// TwinCAT 3 PLC project TE1108
// ProgramVersion: 3.1.4026.22
// libraries:
//   Tc2_EtherCAT, * (Beckhoff Automation GmbH)
//   Tc2_IoFunctions, * (Beckhoff Automation GmbH)
//   Tc2_Standard, * (Beckhoff Automation GmbH)
//   Tc2_System, * (Beckhoff Automation GmbH)
//   Tc2_Utilities, * (Beckhoff Automation GmbH)
//   Tc3_Module, * (Beckhoff Automation GmbH)
// project tree:
//   DUTs/COMPONENTS/CAMERA/ ST_Camera.TcDUT, E_Camera_State.TcDUT, ST_Camera_CycleData.TcDUT (not stored), ST_Camera_CMD.TcDUT (not stored)
//   DUTs/COMPONENTS/GENERIC/ ST_GeneralStationCMD.TcDUT (not stored), ST_StationStatus.TcDUT
//   DUTs/COMPONENTS/HEIGHT TEST/ ST_HeightTest.TcDUT, ST_HeightTest_CMD.TcDUT, ST_ProbesSettings.TcDUT, E_HeightTest_State.TcDUT, ST_HeightTest_CycleData.TcDUT (not stored)
//   DUTs/COMPONENTS/LEAK TESTER/ ST_LeakTester.TcDUT, ST_LeakTester_CMD.TcDUT, E_LeakTester_State.TcDUT (not stored), ST_LeakTester_CycleData.TcDUT (not stored)
//   DUTs/COMPONENTS/MAIN CYLINDER/ ST_ProcessCylinder.TcDUT, E_ProcessCylinder_State.TcDUT, ST_ProcessCylinder_CMD.TcDUT (not stored)
//   DUTs/COMPONENTS/PROCESS DOOR/ E_ProcessDoor_State.TcDUT, ST_ProcessDoor.TcDUT, ST_ProcessDoor_CMD.TcDUT
//   DUTs/COMPONENTS/PUCK_LOCKER/ E_PuckLockerMode.TcDUT, E_PuckLockerState.TcDUT, ST_PuckLocker.TcDUT, ST_PuckLockerHMI.TcDUT
//   DUTs/HMI/ ST_Animations.TcDUT, ST_StatisticsHMI.TcDUT, ST_StatusBanner.TcDUT, ST_Timers.TcDUT (not stored)
//   DUTs/IO/CAMERA/ ST_KeyenceCamera_I_O.TcDUT
//   DUTs/IO/CARDS/ ST_EL1918_C.TcDUT, ST_EL3058.TcDUT (not stored), ST_EL1918_A.TcDUT, ST_EL1918_B.TcDUT, ST_EL2904.TcDUT, ST_EL6910.TcDUT, ST_EL6633.TcDUT, ST_EL9410.TcDUT, ST_K1100.TcDUT (not stored), ST_EL6070.TcDUT (not stored), ST_Terminal_Info.TcDUT (not stored), ST_EL1809.TcDUT, ST_EL2809_A.TcDUT
//   DUTs/IO/LEAK_TESTERS/ ST_General_LeakTester_I_O.TcDUT (not stored), st_i28General_I_O.TcDUT, st_i28LasResult.TcDUT, st_i28LiveMeasurement.TcDUT
//   DUTs/IO/PROBES/ ST_ProbesSet.TcDUT, ST_Probes_I_O.TcDUT
//   DUTs/MASTER/ E_MachineState.TcDUT, ST_ButtonsLamps.TcDUT, ST_HMI_IO.TcDUT (not stored), ST_MACHINE.TcDUT, ST_MachineStatus.TcDUT, ST_MasterCTRL.TcDUT, ST_Puls.TcDUT
//   DUTs/MASTER/log_CSV/ ST_TableCycleData.TcDUT (not stored), ST_UserLog.TcDUT, ST_CycleData.TcDUT (not stored)
//   DUTs/MASTER/PROCESS CYCLES/ E_General_ProcessCycle.TcDUT
//   DUTs/PDFMaker/ ST_EventsPDF.TcDUT (not stored), ST_EventsPdfConstants.TcDUT (not stored), ST_JavasCriptPDF.TcDUT (not stored), ST_PDFMaker.TcDUT (not stored)
//   DUTs/ ST_SafeOutputsReading.TcDUT (not stored), ST_TwinSAFE.TcDUT
//   DUTs/USER_ALARMS_EVENTS/EVENTS/ ST_ActiveEvents.TcDUT, ST_EventsAssigment.TcDUT, ST_EventsAssigmentGeneral.TcDUT, ST_EventsHistory.TcDUT (not stored), ST_EVENT.TcDUT, ST_StationEvents.TcDUT
//   DUTs/USER_ALARMS_EVENTS/ ST_UserLogHMI.TcDUT
//   GVLs/ GVL_Constants.TcGVL (not stored), GVL_HMI.TcGVL, GVL_IO.TcGVL, GVL_Master.TcGVL, GVL_Persistent.TcGVL (not stored), GVL_Stations.TcGVL
//   / PlcTask.TcTTO
//   POUs/A_MASTER/ A_1_PRG_Main_Master.TcPOU, A_2_PRG_MachineCtrl.TcPOU, A_3_PRG_FaultHandling.TcPOU
//   POUs/B_STATIONS/B_1_LEAK_TEST/ B_1_1_PRG_Master_Leak_Test.TcPOU
//   POUs/B_STATIONS/B_2_HEIGHT_TEST/ B_2_1_PRG_Master_Height_Test.TcPOU
//   POUs/B_STATIONS/B_3_CAMERA/ B_3_1_PRG_Master_Camera.TcPOU
//   POUs/B_STATIONS/B_4_PROCESS_CYLINDER__SLIDE_DOOR/ B_4_1_PRG_Master_ProcessCylinder.TcPOU, B_4_2_PRG_Master_ProcessDoor.TcPOU
//   POUs/B_STATIONS/B_5_PUCK_LOCKER/ B_5_1_PRG_PuckLocker.TcPOU
//   POUs/C_HMI/ C_1_PRG_MainHMI.TcPOU
//   POUs/D_CSV/ D_1_PRG_CycleDataCSV.TcPOU
//   POUs/ MAIN.TcPOU (not stored)
//   POUs/Utilities/ FB_EventsManager.TcPOU (not stored), FB_PDFMaker.TcPOU (not stored), FB_Scale.TcPOU, FB_UserLog.TcPOU (not stored), FB_Pulse.TcPOU, FB_TerminalInfo.TcPOU (not stored), FB_TimeControl.TcPOU (not stored), PRG_Puls.TcPOU
// real-time tasks:
//   TASK PlcTask: cycle T#10ms, priority 20, ADS port 350
// I/O:
//   DEVICE Device1(EtherCAT), AmsNetId 192.168.7.156.4.1
//     Term 1 (EK1100) [EK1100 EtherCAT Coupler (2A E-Bus)]
//       Term 2 (EL6070-0033) [EL6070-0033 1Ch. Licence key terminal, individual licences]
//       Term 3 (EL6910) [EL6910, TwinSAFE PLC]
//       Term 4 (EL1918) [EL1918, 8Ch. Safety Input 24V, TwinSAFE]
//         modules: Module 1 (FSOE), Module 2 (FSLOGIC)
//       Term 5 (EL1918) [EL1918, 8Ch. Safety Input 24V, TwinSAFE]
//         modules: Module 1 (FSOE), Module 2 (FSLOGIC)
//       Term 6 (EL2904) [EL2904, 4 Ch. Safety Output 24V, 0.5A, TwinSAFE]
//         modules: Module 1 (FSOES), Module 2 (DO)
//       Term 7 (EL9410) [EL9410 E-Bus Power Supplier  (Diagnostics)]
//       Term 8 (EL1809) [EL1809 16Ch. Dig. Input 24V, 3ms]
//       Term 9 (EL2809) [EL2809 16Ch. Dig. Output 24V, 0.5A]
//       Term 10 (EL3058) [EL3058 8Ch. Ana. Input 4-20mA]
//       Term 11 (EL1918) [EL1918, 8Ch. Safety Input 24V, TwinSAFE]
//         modules: Module 1 (FSOE), Module 2 (FSLOGIC)
//       Term 12 (EL6633) [EL6633 PROFINET IO Controller]
//       Term 13 (EL9011) [EL9011 End Terminal]
//     Box 21 (DL-EC1A) [DL-EC1A]
//   DEVICE Profinet1 (EL6633), AmsNetId 192.168.7.156.2.1
//     camera-4 [KEYENCE CORPORATION. IV4-XXXX IV4-XXXX] (disabled)
//       modules: Term 7 (DAP Module), Term 8 (Command Control), Term 9 (Additional Setting Value), Term 10 (Command Status Bits), Term 11 (Device Result Bits), Term 12 (Device Status Words), Term 13 (Device Statistics), Term 14 (Position Adjust Result), Term 15 (Tool Result), Term 16 (Tool Result), Term 17 (Tool Result), Term 18 (Tool Result), Term 19 (Tool Result)
//     camera-3 [KEYENCE CORPORATION. IV4-XXXX IV4-XXXX] (disabled)
//       modules: Term 20 (DAP Module), Term 21 (Command Control), Term 22 (Additional Setting Value), Term 23 (Command Status Bits), Term 24 (Device Result Bits), Term 25 (Device Status Words), Term 26 (Device Statistics), Term 27 (Position Adjust Result), Term 28 (Tool Result), Term 29 (Tool Result), Term 30 (Tool Result), Term 31 (Tool Result), Term 32 (Tool Result)
//     camera-1 [KEYENCE CORPORATION. IV4-XXXX IV4-XXXX]
//       modules: Term 93 (DAP Module), Term 94 (Command Control), Term 95 (Additional Setting Value), Term 96 (Command Status Bits), Term 97 (Device Result Bits), Term 98 (Device Status Words), Term 99 (Device Statistics), Term 100 (Position Adjust Result), Term 101 (Tool Result), Term 102 (Tool Result), Term 103 (Tool Result), Term 104 (Tool Result), Term 105 (Tool Result)
//     camera-2 [KEYENCE CORPORATION. IV4-XXXX IV4-XXXX]
//       modules: Term 166 (DAP Module), Term 167 (Command Control), Term 168 (Additional Setting Value), Term 169 (Command Status Bits), Term 170 (Device Result Bits), Term 171 (Device Status Words), Term 172 (Device Statistics), Term 173 (Position Adjust Result), Term 174 (Tool Result), Term 175 (Tool Result), Term 176 (Tool Result), Term 177 (Tool Result), Term 178 (Tool Result)
//     fpc1 [Cincinnati Test Systems 1-port Device 00210]
//       modules: Term 1 (DAP Module), Term 2 (PLC Input), Term 3 (PLC Output  )
//     fpc2 [Cincinnati Test Systems 1-port Device 00210]
//       modules: Term 4 (DAP Module), Term 5 (PLC Input), Term 6 (PLC Output  )
// variable links:
//   Device1(EtherCAT) <-> Device1(EtherCAT)/Term 1 (EK1100)/Term 11 (EL1918)
//     Term 1 (EK1100)/Term 3 (EL6910)/ConnectionInputs/Message_38 TxPDO <-> Module 1 (FSOE)/FSoE Outputs/FSOE
//     Term 1 (EK1100)/Term 3 (EL6910)/ConnectionOutputs/Message_38 RxPDO <-> Module 1 (FSOE)/FSoE Inputs/FSOE
//   Device1(EtherCAT) <-> Device1(EtherCAT)/Term 1 (EK1100)/Term 4 (EL1918)
//     Term 1 (EK1100)/Term 3 (EL6910)/ConnectionInputs/Message_8 TxPDO <-> Module 1 (FSOE)/FSoE Outputs/FSOE
//     Term 1 (EK1100)/Term 3 (EL6910)/ConnectionOutputs/Message_8 RxPDO <-> Module 1 (FSOE)/FSoE Inputs/FSOE
//   Device1(EtherCAT) <-> Device1(EtherCAT)/Term 1 (EK1100)/Term 5 (EL1918)
//     Term 1 (EK1100)/Term 3 (EL6910)/ConnectionInputs/Message_9 TxPDO <-> Module 1 (FSOE)/FSoE Outputs/FSOE
//     Term 1 (EK1100)/Term 3 (EL6910)/ConnectionOutputs/Message_9 RxPDO <-> Module 1 (FSOE)/FSoE Inputs/FSOE
//   Device1(EtherCAT) <-> Device1(EtherCAT)/Term 1 (EK1100)/Term 6 (EL2904)
//     Term 1 (EK1100)/Term 3 (EL6910)/ConnectionInputs/Message_10 TxPDO <-> Module 1 (FSOES)/RxPDO/FSOE
//     Term 1 (EK1100)/Term 3 (EL6910)/ConnectionOutputs/Message_10 RxPDO <-> Module 1 (FSOES)/TxPDO/FSOE
//   TE1108/TE1108 Instance <-> Device1(EtherCAT)/Box 21 (DL-EC1A)
//     PlcTask Inputs/GVL_IO.Probes.bGeneralError <-> Status of System/Error Status
//     PlcTask Inputs/GVL_IO.Probes.stProbesSet[1].abProbeError[1] <-> ID01 Status/ID01 Error Status
//     PlcTask Inputs/GVL_IO.Probes.stProbesSet[1].abProbeError[2] <-> ID02 Status/ID02 Error Status
//     PlcTask Inputs/GVL_IO.Probes.stProbesSet[1].abProbeError[3] <-> ID03 Status/ID03 Error Status
//     PlcTask Inputs/GVL_IO.Probes.stProbesSet[1].abProbeError[4] <-> ID04 Status/ID04 Error Status
//     PlcTask Inputs/GVL_IO.Probes.stProbesSet[2].abProbeError[1] <-> ID05 Status/ID05 Error Status
//     PlcTask Inputs/GVL_IO.Probes.stProbesSet[2].abProbeError[2] <-> ID06 Status/ID06 Error Status
//     PlcTask Inputs/GVL_IO.Probes.stProbesSet[2].abProbeError[3] <-> ID07 Status/ID07 Error Status
//     PlcTask Inputs/GVL_IO.Probes.stProbesSet[2].abProbeError[4] <-> ID08 Status/ID08 Error Status
//     PlcTask Inputs/GVL_IO.Probes.stProbesSet[1].anRawMeasurement[1] <-> ID01 Current Value/ID01 Current Value (P.V.)
//     PlcTask Inputs/GVL_IO.Probes.stProbesSet[1].anRawMeasurement[2] <-> ID02 Current Value/ID02 Current Value (P.V.)
//     PlcTask Inputs/GVL_IO.Probes.stProbesSet[1].anRawMeasurement[3] <-> ID03 Current Value/ID03 Current Value (P.V.)
//     PlcTask Inputs/GVL_IO.Probes.stProbesSet[1].anRawMeasurement[4] <-> ID04 Current Value/ID04 Current Value (P.V.)
//     PlcTask Inputs/GVL_IO.Probes.stProbesSet[2].anRawMeasurement[1] <-> ID05 Current Value/ID05 Current Value (P.V.)
//     PlcTask Inputs/GVL_IO.Probes.stProbesSet[2].anRawMeasurement[2] <-> ID06 Current Value/ID06 Current Value (P.V.)
//     PlcTask Inputs/GVL_IO.Probes.stProbesSet[2].anRawMeasurement[3] <-> ID07 Current Value/ID07 Current Value (P.V.)
//     PlcTask Inputs/GVL_IO.Probes.stProbesSet[2].anRawMeasurement[4] <-> ID08 Current Value/ID08 Current Value (P.V.)
//     PlcTask Inputs/GVL_IO.Probes.stTerminalInfo.nTerminal_State <-> InfoData/State
//     PlcTask Outputs/GVL_IO.Probes.abPresetProbe <-> Input Request 1/Request 1
//   TE1108/TE1108 Instance <-> Device1(EtherCAT)/Term 1 (EK1100)
//     PlcTask Inputs/GVL_IO.dw_T01_EK1100.stTerminalInfo.nTerminal_State <-> InfoData/State
//   TE1108/TE1108 Instance <-> Device1(EtherCAT)/Term 1 (EK1100)/Term 10 (EL3058)
//     PlcTask Inputs/GVL_IO.dw_T10_EL3058.iMainPressure <-> AI Standard Channel 1/Value
//     PlcTask Inputs/GVL_IO.dw_T10_EL3058.stTerminalInfo.nTerminal_State <-> InfoData/State
//   TE1108/TE1108 Instance <-> Device1(EtherCAT)/Term 1 (EK1100)/Term 11 (EL1918)
//     PlcTask Inputs/GVL_IO.dw_T11_EL1918.iD3ProcessCylinderFeedback <-> Module 1 (FSOE)/FSoE Inputs/FSOE/FSIN Module 3.Input
//     PlcTask Inputs/GVL_IO.dw_T11_EL1918.iD3ProcessCylinderRetracted1 <-> Module 1 (FSOE)/FSoE Inputs/FSOE/FSIN Module 1.Input
//     PlcTask Inputs/GVL_IO.dw_T11_EL1918.iD3ProcessCylinderRetracted2 <-> Module 1 (FSOE)/FSoE Inputs/FSOE/FSIN Module 2.Input
//     PlcTask Inputs/GVL_IO.dw_T11_EL1918.stTerminalInfo.nTerminal_State <-> InfoData/State
//   TE1108/TE1108 Instance <-> Device1(EtherCAT)/Term 1 (EK1100)/Term 12 (EL6633)
//     PlcTask Inputs/GVL_IO.dw_T12_EL6633.stTerminalInfo.nTerminal_State <-> InfoData/State
//   TE1108/TE1108 Instance <-> Device1(EtherCAT)/Term 1 (EK1100)/Term 2 (EL6070-0033)
//     PlcTask Inputs/GVL_IO.dw_T02_EL6070.stTerminalInfo.nTerminal_State <-> InfoData/State
//   TE1108/TE1108 Instance <-> Device1(EtherCAT)/Term 1 (EK1100)/Term 3 (EL6910)
//     PlcTask Inputs/GVL_IO.dw_T03_EL6910.stTerminalInfo.nTerminal_State <-> InfoData/State
//     PlcTask Inputs/GVL_IO.stTwinSAFE.qAirErrorSignal <-> StandardInputs/TwinSafeGroup1.AirErrorSignal_59
//     PlcTask Inputs/GVL_IO.stTwinSAFE.qAirPressureAbove <-> StandardInputs/TwinSafeGroup1.AirPressureAbove_26
//     PlcTask Inputs/GVL_IO.stTwinSAFE.qAirPressureBelow <-> StandardInputs/TwinSafeGroup1.AirPressureBelow_25
//     PlcTask Inputs/GVL_IO.stTwinSAFE.qAirPressureOK <-> StandardInputs/TwinSafeGroup1.AirPressureOK_41
//     PlcTask Inputs/GVL_IO.stTwinSAFE.qComError <-> StandardInputs/TwinSafeGroup1.COMError_74
//     PlcTask Inputs/GVL_IO.stTwinSAFE.qE_StopPressed <-> StandardInputs/TwinSafeGroup1.E_StopPressed_32
//     PlcTask Inputs/GVL_IO.stTwinSAFE.qFBError <-> StandardInputs/TwinSafeGroup1.FBError_73
//     PlcTask Inputs/GVL_IO.stTwinSAFE.qMainDoorOpenned <-> StandardInputs/TwinSafeGroup1.DoorOpenned_68
//     PlcTask Inputs/GVL_IO.stTwinSAFE.qMainDoorUnsafe <-> StandardInputs/TwinSafeGroup1.MainDoorUnsafe_49
//     PlcTask Inputs/GVL_IO.stTwinSAFE.qOtherError <-> StandardInputs/TwinSafeGroup1.OtherError_75
//     PlcTask Inputs/GVL_IO.stTwinSAFE.qProcessCylinderRetracted <-> StandardInputs/TwinSafeGroup1.ProcessCylinderRetracted_60
//     PlcTask Inputs/GVL_IO.stTwinSAFE.qProcessCylinderUnsafe <-> StandardInputs/TwinSafeGroup1.ProcessCylinderUnsafe_54
//     PlcTask Inputs/GVL_IO.stTwinSAFE.qProcessDoorUnSafe <-> StandardInputs/TwinSafeGroup1.ProcessDoorUnsafe_34
//     PlcTask Inputs/GVL_IO.stTwinSAFE.qSafetyOk <-> StandardInputs/TwinSafeGroup1.SafetyOK_30
//     PlcTask Inputs/GVL_IO.stTwinSAFE.qSystemSafe <-> StandardInputs/TwinSafeGroup1.SystemSafe_72
//     PlcTask Inputs/GVL_IO.stTwinSAFE.qTwoHandsSafe <-> StandardInputs/TwinSafeGroup1.TwoHandsSafe_77
//     PlcTask Inputs/GVL_IO.stTwinSAFE.qTwoHandsUnsafe <-> StandardInputs/TwinSafeGroup1.TwoHandsUnsafe_35
//     PlcTask Outputs/GVL_IO.stTwinSAFE.iAirPressureMaxValue <-> StandardOutputs/TwinSafeGroup1.AirPressureMaxVal_23
//     PlcTask Outputs/GVL_IO.stTwinSAFE.iAirPressureMinValue <-> StandardOutputs/TwinSafeGroup1.AirPressureMinVal_22
//     PlcTask Outputs/GVL_IO.stTwinSAFE.iAirSupplyMeasurement <-> StandardOutputs/TwinSafeGroup1.AirSupplyMeasurement_19
//     PlcTask Outputs/GVL_IO.stTwinSAFE.iMachineHoming_Manual <-> StandardOutputs/TwinSafeGroup1.MachineHoming_Manual_78
//     PlcTask Outputs/GVL_IO.stTwinSAFE.iMachineStopped <-> StandardOutputs/TwinSafeGroup1.MachineStopped_70
//     PlcTask Outputs/GVL_IO.stTwinSAFE.iProcessDoorClosedCondition <-> StandardOutputs/TwinSafeGroup1.ProcessDoorClosedCondition_16
//     PlcTask Outputs/GVL_IO.stTwinSAFE.iProcessDoorClosing <-> StandardOutputs/TwinSafeGroup1.ProcessDoor Closing_29
//     PlcTask Outputs/GVL_IO.stTwinSAFE.iRunSafety <-> StandardOutputs/TwinSafeGroup1.RunSafety_69
//     PlcTask Outputs/GVL_IO.stTwinSAFE.iSafetyErrorAcknowledge <-> StandardOutputs/TwinSafeGroup1.SafetyErrorAcknowledge_55
//   TE1108/TE1108 Instance <-> Device1(EtherCAT)/Term 1 (EK1100)/Term 4 (EL1918)
//     PlcTask Inputs/GVL_IO.dw_T04_EL1918.iD1MainDoorFB <-> Module 1 (FSOE)/FSoE Inputs/FSOE/FSIN Module 6.Input
//     PlcTask Inputs/GVL_IO.dw_T04_EL1918.iD1MainDoorLocked1 <-> Module 1 (FSOE)/FSoE Inputs/FSOE/FSIN Module 4.Input
//     PlcTask Inputs/GVL_IO.dw_T04_EL1918.iD1MainDoorLocked2 <-> Module 1 (FSOE)/FSoE Inputs/FSOE/FSIN Module 5.Input
//     PlcTask Inputs/GVL_IO.dw_T04_EL1918.iEStopChannel1 <-> Module 1 (FSOE)/FSoE Inputs/FSOE/FSIN Module 1.Input
//     PlcTask Inputs/GVL_IO.dw_T04_EL1918.iEStopChannel2 <-> Module 1 (FSOE)/FSoE Inputs/FSOE/FSIN Module 2.Input
//     PlcTask Inputs/GVL_IO.dw_T04_EL1918.iFestoMS6DumpValveFB <-> Module 1 (FSOE)/FSoE Inputs/FSOE/FSIN Module 8.Input
//     PlcTask Inputs/GVL_IO.dw_T04_EL1918.iFestoMS6ValveFB <-> Module 1 (FSOE)/FSoE Inputs/FSOE/FSIN Module 7.Input
//     PlcTask Inputs/GVL_IO.dw_T04_EL1918.iResetButton <-> Module 1 (FSOE)/FSoE Inputs/FSOE/FSIN Module 3.Input
//     PlcTask Inputs/GVL_IO.dw_T04_EL1918.stTerminalInfo.nTerminal_State <-> InfoData/State
//   TE1108/TE1108 Instance <-> Device1(EtherCAT)/Term 1 (EK1100)/Term 5 (EL1918)
//     PlcTask Inputs/GVL_IO.dw_T05_EL1918.iLeftTouchButtonNC <-> Module 1 (FSOE)/FSoE Inputs/FSOE/FSIN Module 1.Input
//     PlcTask Inputs/GVL_IO.dw_T05_EL1918.iLeftTouchButtonNO <-> Module 1 (FSOE)/FSoE Inputs/FSOE/FSIN Module 3.Input
//     PlcTask Inputs/GVL_IO.dw_T05_EL1918.iProcessDoorClosed1 <-> Module 1 (FSOE)/FSoE Inputs/FSOE/FSIN Module 5.Input
//     PlcTask Inputs/GVL_IO.dw_T05_EL1918.iProcessDoorClosed2 <-> Module 1 (FSOE)/FSoE Inputs/FSOE/FSIN Module 6.Input
//     PlcTask Inputs/GVL_IO.dw_T05_EL1918.iProcessDoorFB <-> Module 1 (FSOE)/FSoE Inputs/FSOE/FSIN Module 7.Input
//     PlcTask Inputs/GVL_IO.dw_T05_EL1918.iRightTouchButtonNC <-> Module 1 (FSOE)/FSoE Inputs/FSOE/FSIN Module 2.Input
//     PlcTask Inputs/GVL_IO.dw_T05_EL1918.iRightTouchButtonNO <-> Module 1 (FSOE)/FSoE Inputs/FSOE/FSIN Module 4.Input
//     PlcTask Inputs/GVL_IO.dw_T05_EL1918.stTerminalInfo.nTerminal_State <-> InfoData/State
//   TE1108/TE1108 Instance <-> Device1(EtherCAT)/Term 1 (EK1100)/Term 6 (EL2904)
//     PlcTask Inputs/GVL_IO.dw_T06_EL2904.stTerminalInfo.nTerminal_State <-> InfoData/State
//   TE1108/TE1108 Instance <-> Device1(EtherCAT)/Term 1 (EK1100)/Term 7 (EL9410)
//     PlcTask Inputs/GVL_IO.dw_T07_EL9410.stTerminalInfo.nTerminal_State <-> InfoData/State
//   TE1108/TE1108 Instance <-> Device1(EtherCAT)/Term 1 (EK1100)/Term 8 (EL1809)
//     PlcTask Inputs/GVL_IO.dw_T08_EL1809.iPartPresentNest1 <-> Channel 5/Input
//     PlcTask Inputs/GVL_IO.dw_T08_EL1809.iPartPresentNest2 <-> Channel 6/Input
//     PlcTask Inputs/GVL_IO.dw_T08_EL1809.iProcessCylinderExtended <-> Channel 10/Input
//     PlcTask Inputs/GVL_IO.dw_T08_EL1809.iPuckSensorDown <-> Channel 16/Input
//     PlcTask Inputs/GVL_IO.dw_T08_EL1809.iPuckSensorUp <-> Channel 15/Input
//     PlcTask Inputs/GVL_IO.dw_T08_EL1809.iRejectSensor <-> Channel 11/Input
//     PlcTask Inputs/GVL_IO.dw_T08_EL1809.iStartButoon <-> Channel 1/Input
//     PlcTask Inputs/GVL_IO.dw_T08_EL1809.iStopButton <-> Channel 2/Input
//     PlcTask Inputs/GVL_IO.dw_T08_EL1809.iUP_OK <-> Channel 3/Input
//     PlcTask Inputs/GVL_IO.dw_T08_EL1809.iUS_OK <-> Channel 4/Input
//     PlcTask Inputs/GVL_IO.dw_T08_EL1809.stTerminalInfo.nTerminal_State <-> InfoData/State
//   TE1108/TE1108 Instance <-> Device1(EtherCAT)/Term 1 (EK1100)/Term 9 (EL2809)
//     PlcTask Inputs/GVL_IO.dw_T09_EL2809.stTerminalInfo.nTerminal_State <-> InfoData/State
//     PlcTask Outputs/GVL_IO.dw_T09_EL2809.qCloseProcessDoor <-> Channel 4/Output
//     PlcTask Outputs/GVL_IO.dw_T09_EL2809.qExtendProcessCylinder <-> Channel 6/Output
//     PlcTask Outputs/GVL_IO.dw_T09_EL2809.qIndicatorLED1_Green <-> Channel 9/Output
//     PlcTask Outputs/GVL_IO.dw_T09_EL2809.qIndicatorLED2_Green <-> Channel 11/Output
//     PlcTask Outputs/GVL_IO.dw_T09_EL2809.qIndicatorLED1_Red <-> Channel 8/Output
//     PlcTask Outputs/GVL_IO.dw_T09_EL2809.qIndicatorLED2_Red <-> Channel 10/Output
//     PlcTask Outputs/GVL_IO.dw_T09_EL2809.qOpenProcessDoor <-> Channel 3/Output
//     PlcTask Outputs/GVL_IO.dw_T09_EL2809.qPanelLightLED <-> Channel 7/Output
//     PlcTask Outputs/GVL_IO.dw_T09_EL2809.qPuckLockerPinCommand <-> Channel 16/Output
//     PlcTask Outputs/GVL_IO.dw_T09_EL2809.qResetButtonLED <-> Channel 2/Output
//     PlcTask Outputs/GVL_IO.dw_T09_EL2809.qRetractProcessCylinder <-> Channel 5/Output
//     PlcTask Outputs/GVL_IO.dw_T09_EL2809.qStartButtonLED <-> Channel 1/Output
//   TE1108/TE1108 Instance <-> Profinet1 (EL6633)/camera-1
//     PlcTask Inputs/GVL_IO.Camera1_IO.bAlarm <-> API/Term 96 (Command Status Bits)/Subterm 112 (Command Status Bits)/Inputs/Command Status Bits Register3/Warning
//     PlcTask Inputs/GVL_IO.Camera1_IO.bBusy <-> API/Term 96 (Command Status Bits)/Subterm 112 (Command Status Bits)/Inputs/Command Status Bits Register2/Busy
//     PlcTask Inputs/GVL_IO.Camera1_IO.bError <-> API/Term 96 (Command Status Bits)/Subterm 112 (Command Status Bits)/Inputs/Command Status Bits Register3/Error
//     PlcTask Inputs/GVL_IO.Camera1_IO.bReady <-> API/Term 96 (Command Status Bits)/Subterm 112 (Command Status Bits)/Inputs/Command Status Bits Register2/Ready
//     PlcTask Inputs/GVL_IO.Camera1_IO.bResultReady <-> API/Term 96 (Command Status Bits)/Subterm 112 (Command Status Bits)/Inputs/Command Status Bits Register2/Result_Ready
//     PlcTask Inputs/GVL_IO.Camera1_IO.bRun <-> API/Term 96 (Command Status Bits)/Subterm 112 (Command Status Bits)/Inputs/Command Status Bits Register2/Run
//     PlcTask Inputs/GVL_IO.Camera1_IO.bTotalResult <-> API/Term 97 (Device Result Bits)/Subterm 113 (Device Result Bits)/Inputs/Device Result Bits Register0/Total_Status
//     PlcTask Inputs/GVL_IO.Camera1_IO.bTriggerFail <-> API/Term 96 (Command Status Bits)/Subterm 112 (Command Status Bits)/Inputs/Command Status Bits Register1/Trigger_Fail
//     PlcTask Inputs/GVL_IO.Camera1_IO.nScore <-> API/Term 101 (Tool Result)/Subterm 117 (Tool Result)/Inputs/Score
//     PlcTask Outputs/GVL_IO.Camera1_IO.bClearBuffer <-> API/Term 94 (Command Control)/Subterm 110 (Command Control)/Outputs/Command Control Register0/Clear_Buffer
//     PlcTask Outputs/GVL_IO.Camera1_IO.bReset <-> API/Term 94 (Command Control)/Subterm 110 (Command Control)/Outputs/Command Control Register0/Clear_Warning
//     PlcTask Outputs/GVL_IO.Camera1_IO.bResetStatistics <-> API/Term 94 (Command Control)/Subterm 110 (Command Control)/Outputs/Command Control Register0/Reset_Statistics
//     PlcTask Outputs/GVL_IO.Camera1_IO.bResultReadyAck <-> API/Term 94 (Command Control)/Subterm 110 (Command Control)/Outputs/Command Control Register1/Result_Ready_Ack
//     PlcTask Outputs/GVL_IO.Camera1_IO.bSetTreshold <-> API/Term 94 (Command Control)/Subterm 110 (Command Control)/Outputs/Command Control Register0/Set_Threshold
//     PlcTask Outputs/GVL_IO.Camera1_IO.bSettingNo <-> API/Term 94 (Command Control)/Subterm 110 (Command Control)/Outputs/Setting No.
//     PlcTask Outputs/GVL_IO.Camera1_IO.bSettingVal <-> API/Term 94 (Command Control)/Subterm 110 (Command Control)/Outputs/Setting Value1
//     PlcTask Outputs/GVL_IO.Camera1_IO.bTrigger <-> API/Term 94 (Command Control)/Subterm 110 (Command Control)/Outputs/Command Control Register0/Trigger
//   TE1108/TE1108 Instance <-> Profinet1 (EL6633)/camera-2
//     PlcTask Inputs/GVL_IO.Camera2_IO.bAlarm <-> API/Term 169 (Command Status Bits)/Subterm 187 (Command Status Bits)/Inputs/Command Status Bits Register3/Warning
//     PlcTask Inputs/GVL_IO.Camera2_IO.bBusy <-> API/Term 169 (Command Status Bits)/Subterm 187 (Command Status Bits)/Inputs/Command Status Bits Register2/Busy
//     PlcTask Inputs/GVL_IO.Camera2_IO.bError <-> API/Term 169 (Command Status Bits)/Subterm 187 (Command Status Bits)/Inputs/Command Status Bits Register3/Error
//     PlcTask Inputs/GVL_IO.Camera2_IO.bReady <-> API/Term 169 (Command Status Bits)/Subterm 187 (Command Status Bits)/Inputs/Command Status Bits Register2/Ready
//     PlcTask Inputs/GVL_IO.Camera2_IO.bResultReady <-> API/Term 169 (Command Status Bits)/Subterm 187 (Command Status Bits)/Inputs/Command Status Bits Register2/Result_Ready
//     PlcTask Inputs/GVL_IO.Camera2_IO.bRun <-> API/Term 169 (Command Status Bits)/Subterm 187 (Command Status Bits)/Inputs/Command Status Bits Register2/Run
//     PlcTask Inputs/GVL_IO.Camera2_IO.bTotalResult <-> API/Term 170 (Device Result Bits)/Subterm 188 (Device Result Bits)/Inputs/Device Result Bits Register0/Total_Status
//     PlcTask Inputs/GVL_IO.Camera2_IO.bTriggerFail <-> API/Term 169 (Command Status Bits)/Subterm 187 (Command Status Bits)/Inputs/Command Status Bits Register1/Trigger_Fail
//     PlcTask Inputs/GVL_IO.Camera2_IO.nScore <-> API/Term 174 (Tool Result)/Subterm 192 (Tool Result)/Inputs/Score
//     PlcTask Outputs/GVL_IO.Camera2_IO.bClearBuffer <-> API/Term 167 (Command Control)/Subterm 185 (Command Control)/Outputs/Command Control Register0/Clear_Buffer
//     PlcTask Outputs/GVL_IO.Camera2_IO.bReset <-> API/Term 167 (Command Control)/Subterm 185 (Command Control)/Outputs/Command Control Register0/Clear_Warning
//     PlcTask Outputs/GVL_IO.Camera2_IO.bResetStatistics <-> API/Term 167 (Command Control)/Subterm 185 (Command Control)/Outputs/Command Control Register0/Reset_Statistics
//     PlcTask Outputs/GVL_IO.Camera2_IO.bResultReadyAck <-> API/Term 167 (Command Control)/Subterm 185 (Command Control)/Outputs/Command Control Register1/Result_Ready_Ack
//     PlcTask Outputs/GVL_IO.Camera2_IO.bSetTreshold <-> API/Term 167 (Command Control)/Subterm 185 (Command Control)/Outputs/Command Control Register0/Set_Threshold
//     PlcTask Outputs/GVL_IO.Camera2_IO.bSettingNo <-> API/Term 167 (Command Control)/Subterm 185 (Command Control)/Outputs/Setting No.
//     PlcTask Outputs/GVL_IO.Camera2_IO.bSettingVal <-> API/Term 167 (Command Control)/Subterm 185 (Command Control)/Outputs/Setting Value1
//     PlcTask Outputs/GVL_IO.Camera2_IO.bTrigger <-> API/Term 167 (Command Control)/Subterm 185 (Command Control)/Outputs/Command Control Register0/Trigger
//   TE1108/TE1108 Instance <-> Profinet1 (EL6633)/camera-3
//     PlcTask Inputs/GVL_IO.Camera3_IO.bAlarm <-> API/Term 23 (Command Status Bits)/Subterm 37 (Command Status Bits)/Inputs/Command Status Bits Register3/Warning
//     PlcTask Inputs/GVL_IO.Camera3_IO.bBusy <-> API/Term 23 (Command Status Bits)/Subterm 37 (Command Status Bits)/Inputs/Command Status Bits Register2/Busy
//     PlcTask Inputs/GVL_IO.Camera3_IO.bError <-> API/Term 23 (Command Status Bits)/Subterm 37 (Command Status Bits)/Inputs/Command Status Bits Register3/Error
//     PlcTask Inputs/GVL_IO.Camera3_IO.bReady <-> API/Term 23 (Command Status Bits)/Subterm 37 (Command Status Bits)/Inputs/Command Status Bits Register2/Ready
//     PlcTask Inputs/GVL_IO.Camera3_IO.bResultReady <-> API/Term 23 (Command Status Bits)/Subterm 37 (Command Status Bits)/Inputs/Command Status Bits Register2/Result_Ready
//     PlcTask Inputs/GVL_IO.Camera3_IO.bRun <-> API/Term 23 (Command Status Bits)/Subterm 37 (Command Status Bits)/Inputs/Command Status Bits Register2/Run
//     PlcTask Inputs/GVL_IO.Camera3_IO.bTotalResult <-> API/Term 24 (Device Result Bits)/Subterm 38 (Device Result Bits)/Inputs/Device Result Bits Register0/Total_Status
//     PlcTask Inputs/GVL_IO.Camera3_IO.bTriggerFail <-> API/Term 23 (Command Status Bits)/Subterm 37 (Command Status Bits)/Inputs/Command Status Bits Register1/Trigger_Fail
//     PlcTask Inputs/GVL_IO.Camera3_IO.nScore <-> API/Term 28 (Tool Result)/Subterm 42 (Tool Result)/Inputs/Score
//     PlcTask Outputs/GVL_IO.Camera3_IO.bClearBuffer <-> API/Term 21 (Command Control)/Subterm 35 (Command Control)/Outputs/Command Control Register0/Clear_Buffer
//     PlcTask Outputs/GVL_IO.Camera3_IO.bReset <-> API/Term 21 (Command Control)/Subterm 35 (Command Control)/Outputs/Command Control Register0/Clear_Warning
//     PlcTask Outputs/GVL_IO.Camera3_IO.bResetStatistics <-> API/Term 21 (Command Control)/Subterm 35 (Command Control)/Outputs/Command Control Register0/Reset_Statistics
//     PlcTask Outputs/GVL_IO.Camera3_IO.bResultReadyAck <-> API/Term 21 (Command Control)/Subterm 35 (Command Control)/Outputs/Command Control Register1/Result_Ready_Ack
//     PlcTask Outputs/GVL_IO.Camera3_IO.bSetTreshold <-> API/Term 21 (Command Control)/Subterm 35 (Command Control)/Outputs/Command Control Register0/Set_Threshold
//     PlcTask Outputs/GVL_IO.Camera3_IO.bSettingNo <-> API/Term 21 (Command Control)/Subterm 35 (Command Control)/Outputs/Setting No.
//     PlcTask Outputs/GVL_IO.Camera3_IO.bSettingVal <-> API/Term 21 (Command Control)/Subterm 35 (Command Control)/Outputs/Setting Value1
//     PlcTask Outputs/GVL_IO.Camera3_IO.bTrigger <-> API/Term 21 (Command Control)/Subterm 35 (Command Control)/Outputs/Command Control Register0/Trigger
//   TE1108/TE1108 Instance <-> Profinet1 (EL6633)/camera-4
//     PlcTask Inputs/GVL_IO.Camera4_IO.bAlarm <-> API/Term 10 (Command Status Bits)/Subterm 22 (Command Status Bits)/Inputs/Command Status Bits Register3/Warning
//     PlcTask Inputs/GVL_IO.Camera4_IO.bBusy <-> API/Term 10 (Command Status Bits)/Subterm 22 (Command Status Bits)/Inputs/Command Status Bits Register2/Busy
//     PlcTask Inputs/GVL_IO.Camera4_IO.bError <-> API/Term 10 (Command Status Bits)/Subterm 22 (Command Status Bits)/Inputs/Command Status Bits Register3/Error
//     PlcTask Inputs/GVL_IO.Camera4_IO.bReady <-> API/Term 10 (Command Status Bits)/Subterm 22 (Command Status Bits)/Inputs/Command Status Bits Register2/Ready
//     PlcTask Inputs/GVL_IO.Camera4_IO.bResultReady <-> API/Term 10 (Command Status Bits)/Subterm 22 (Command Status Bits)/Inputs/Command Status Bits Register2/Result_Ready
//     PlcTask Inputs/GVL_IO.Camera4_IO.bRun <-> API/Term 10 (Command Status Bits)/Subterm 22 (Command Status Bits)/Inputs/Command Status Bits Register2/Run
//     PlcTask Inputs/GVL_IO.Camera4_IO.bTotalResult <-> API/Term 11 (Device Result Bits)/Subterm 23 (Device Result Bits)/Inputs/Device Result Bits Register0/Total_Status
//     PlcTask Inputs/GVL_IO.Camera4_IO.bTriggerFail <-> API/Term 10 (Command Status Bits)/Subterm 22 (Command Status Bits)/Inputs/Command Status Bits Register1/Trigger_Fail
//     PlcTask Inputs/GVL_IO.Camera4_IO.nScore <-> API/Term 15 (Tool Result)/Subterm 27 (Tool Result)/Inputs/Score
//     PlcTask Outputs/GVL_IO.Camera4_IO.bClearBuffer <-> API/Term 8 (Command Control)/Subterm 20 (Command Control)/Outputs/Command Control Register0/Clear_Buffer
//     PlcTask Outputs/GVL_IO.Camera4_IO.bReset <-> API/Term 8 (Command Control)/Subterm 20 (Command Control)/Outputs/Command Control Register0/Clear_Warning
//     PlcTask Outputs/GVL_IO.Camera4_IO.bResetStatistics <-> API/Term 8 (Command Control)/Subterm 20 (Command Control)/Outputs/Command Control Register0/Reset_Statistics
//     PlcTask Outputs/GVL_IO.Camera4_IO.bResultReadyAck <-> API/Term 8 (Command Control)/Subterm 20 (Command Control)/Outputs/Command Control Register1/Result_Ready_Ack
//     PlcTask Outputs/GVL_IO.Camera4_IO.bSetTreshold <-> API/Term 8 (Command Control)/Subterm 20 (Command Control)/Outputs/Command Control Register0/Set_Threshold
//     PlcTask Outputs/GVL_IO.Camera4_IO.bSettingNo <-> API/Term 8 (Command Control)/Subterm 20 (Command Control)/Outputs/Setting No.
//     PlcTask Outputs/GVL_IO.Camera4_IO.bSettingVal <-> API/Term 8 (Command Control)/Subterm 20 (Command Control)/Outputs/Setting Value1
//     PlcTask Outputs/GVL_IO.Camera4_IO.bTrigger <-> API/Term 8 (Command Control)/Subterm 20 (Command Control)/Outputs/Command Control Register0/Trigger
//   TE1108/TE1108 Instance <-> Profinet1 (EL6633)/fpc1
//     PlcTask Inputs/GVL_IO.LeakTester1_IO.sti28General_I_O.bInstrumentReady <-> API/Term 2 (PLC Input)/Subterm 4 (Instrument Status)/Inputs/Instrument Status/Instrument_Ready
//     PlcTask Inputs/GVL_IO.LeakTester1_IO.sti28General_I_O.bMalfunction <-> API/Term 2 (PLC Input)/Subterm 4 (Instrument Status)/Inputs/Instrument Status/Malfunction
//     PlcTask Inputs/GVL_IO.LeakTester1_IO.sti28General_I_O.bProgramAccept <-> API/Term 2 (PLC Input)/Subterm 4 (Instrument Status)/Inputs/Instrument Status/Program_Accept
//     PlcTask Inputs/GVL_IO.LeakTester1_IO.sti28General_I_O.bProgramReject <-> API/Term 2 (PLC Input)/Subterm 4 (Instrument Status)/Inputs/Instrument Status/Program_Reject
//     PlcTask Inputs/GVL_IO.LeakTester1_IO.sti28General_I_O.bTestActiveLiveData <-> API/Term 2 (PLC Input)/Subterm 4 (Instrument Status)/Inputs/Instrument Status/Test_Active_Live_Data
//     PlcTask Outputs/GVL_IO.LeakTester1_IO.sti28General_I_O.bReset <-> API/Term 3 (PLC Output  )/Subterm 7 (Instrument Control )/Outputs/Instrument Control/Reset
//     PlcTask Outputs/GVL_IO.LeakTester1_IO.sti28General_I_O.bStart <-> API/Term 3 (PLC Output  )/Subterm 7 (Instrument Control )/Outputs/Instrument Control/Start
//     PlcTask Outputs/GVL_IO.LeakTester1_IO.sti28General_I_O.bStop <-> API/Term 3 (PLC Output  )/Subterm 7 (Instrument Control )/Outputs/Instrument Control/Stop
//   TE1108/TE1108 Instance <-> Profinet1 (EL6633)/fpc2
//     PlcTask Inputs/GVL_IO.LeakTester2_IO.sti28General_I_O.bInstrumentReady <-> API/Term 5 (PLC Input)/Subterm 12 (Instrument Status)/Inputs/Instrument Status/Instrument_Ready
//     PlcTask Inputs/GVL_IO.LeakTester2_IO.sti28General_I_O.bMalfunction <-> API/Term 5 (PLC Input)/Subterm 12 (Instrument Status)/Inputs/Instrument Status/Malfunction
//     PlcTask Inputs/GVL_IO.LeakTester2_IO.sti28General_I_O.bProgramAccept <-> API/Term 5 (PLC Input)/Subterm 12 (Instrument Status)/Inputs/Instrument Status/Program_Accept
//     PlcTask Inputs/GVL_IO.LeakTester2_IO.sti28General_I_O.bProgramReject <-> API/Term 5 (PLC Input)/Subterm 12 (Instrument Status)/Inputs/Instrument Status/Program_Reject
//     PlcTask Inputs/GVL_IO.LeakTester2_IO.sti28General_I_O.bTestActiveLiveData <-> API/Term 5 (PLC Input)/Subterm 12 (Instrument Status)/Inputs/Instrument Status/Test_Active_Live_Data
//     PlcTask Outputs/GVL_IO.LeakTester2_IO.sti28General_I_O.bReset <-> API/Term 6 (PLC Output  )/Subterm 15 (Instrument Control )/Outputs/Instrument Control/Reset
//     PlcTask Outputs/GVL_IO.LeakTester2_IO.sti28General_I_O.bStart <-> API/Term 6 (PLC Output  )/Subterm 15 (Instrument Control )/Outputs/Instrument Control/Start
//     PlcTask Outputs/GVL_IO.LeakTester2_IO.sti28General_I_O.bStop <-> API/Term 6 (PLC Output  )/Subterm 15 (Instrument Control )/Outputs/Instrument Control/Stop

CONFIGURATION TE1108
    RESOURCE PLC ON TwinCAT3
        TASK PlcTask(INTERVAL := T#10ms, PRIORITY := 20);
        PROGRAM MAIN WITH PlcTask : MAIN;
    END_RESOURCE
END_CONFIGURATION

// ---- DUTs/COMPONENTS/CAMERA/ST_Camera.TcDUT
TYPE ST_Camera :
STRUCT
	
	State								: E_Camera_State;
	CMD									: ST_GeneralStationCMD;
	Status								: ST_StationStatus;

END_STRUCT
END_TYPE

// ---- DUTs/COMPONENTS/GENERIC/ST_StationStatus.TcDUT
TYPE ST_StationStatus :
STRUCT
//Universal Module STATUS Struct

	bReady        			:BOOL;	// Module initialized and ready for CMD
    bBusy         			:BOOL;	// Module is busy processing a request
    bDone         			:BOOL;	// Operation successfully completed
	bStopped				:BOOL;	// Station stopped
    bError        			:BOOL;	// Error occurred
    nErrorID      			:INT;	// Error code (ideally enum-based)


	nCurrentTaskID			:UINT;	// Current Task ID
    nCurrentState 			:UINT;	// Current State


	

//-----------------------------------------------------------------------------------------oldschoo1	


END_STRUCT
END_TYPE

// ---- DUTs/COMPONENTS/HEIGHT TEST/ST_HeightTest.TcDUT
TYPE ST_HeightTest :
STRUCT
	
	State						: E_HeightTest_State;
	CMD							: ST_GeneralStationCMD;	
	Status						: ST_StationStatus;
	
END_STRUCT
END_TYPE

// ---- DUTs/COMPONENTS/HEIGHT TEST/ST_HeightTest_CMD.TcDUT
TYPE ST_HeightTest_CMD :
STRUCT
	
	Measurement1			: BOOL;		
	Measurement2			: BOOL;		
	
END_STRUCT
END_TYPE

// ---- DUTs/COMPONENTS/HEIGHT TEST/ST_ProbesSettings.TcDUT
TYPE ST_ProbesSettings :
STRUCT
	
	anDistanceCalibrationBlock			: ARRAY [1..3] OF REAL;	
	nDistanceOffset1					: ARRAY [1..3] OF REAL; 
	nDistanceOffset2					: ARRAY [1..3] OF REAL;
	(*Renan Added 30Jun26 - Nests offset*)
	anNestOffsetByProbe1         		: ARRAY [1..4] OF REAL;
    anNestOffsetByProbe2         		: ARRAY [1..4] OF REAL;
	(*/Renan Added 30Jun26*)	
	anExpectedDistances					: ARRAY [1..3] OF REAL;
	anHeightSetByCalibration1			: ARRAY [1..4] OF REAL;	
	anHeightSetByCalibration2			: ARRAY [1..4] OF REAL;	
	anTolerances						: ARRAY [1..3] OF REAL;	


END_STRUCT
END_TYPE

// ---- DUTs/COMPONENTS/LEAK TESTER/ST_LeakTester.TcDUT
TYPE ST_LeakTester :
STRUCT
	
	State							: E_LeakTester_State;	
	CMD								: ST_GeneralStationCMD;
	Status							: ST_StationStatus;
	
END_STRUCT
END_TYPE

// ---- DUTs/COMPONENTS/LEAK TESTER/ST_LeakTester_CMD.TcDUT
TYPE ST_LeakTester_CMD :
STRUCT
	
	RunLeakTester1		: BOOL;		
	RunLeakTester2		: BOOL;	
	
END_STRUCT
END_TYPE

// ---- DUTs/COMPONENTS/MAIN CYLINDER/ST_ProcessCylinder.TcDUT
TYPE ST_ProcessCylinder :
STRUCT
	
	State						: E_ProcessCylinder_State;
	CMD							: ST_GeneralStationCMD;
	Status						: ST_StationStatus;

END_STRUCT
END_TYPE

// ---- DUTs/COMPONENTS/PROCESS DOOR/E_ProcessDoor_State.TcDUT
{attribute 'qualified_only'}
{attribute 'strict'}
TYPE E_ProcessDoor_State :
(
		//GENERIC
	ABORTED				,
	HOMING				,
	READY				,
	MANUAL_MODE			,
	STOPPING			,
	//SPECIFIC FOR EVERY STATION
	OPEN,
	CLOSE,
	DONE				,
	RESET				
);
END_TYPE

// ---- DUTs/COMPONENTS/PROCESS DOOR/ST_ProcessDoor.TcDUT
TYPE ST_ProcessDoor :
STRUCT
	
	State					: E_ProcessDoor_State;
	CMD						: ST_GeneralStationCMD;
	Status					: ST_StationStatus;

END_STRUCT
END_TYPE

// ---- DUTs/COMPONENTS/PROCESS DOOR/ST_ProcessDoor_CMD.TcDUT
TYPE ST_ProcessDoor_CMD :
STRUCT
	
	OpenDoor					: BOOL;				
	CloseDoor					: BOOL;		
	
END_STRUCT
END_TYPE

// ---- DUTs/COMPONENTS/PUCK_LOCKER/E_PuckLockerMode.TcDUT
{attribute 'qualified_only'}
{attribute 'strict'}
{attribute 'to_string'}
TYPE E_PuckLockerMode :
(
	Disabled := 0,
    Enabled := 1,
    EnabledWithEmptyPuckBypass := 2
);
END_TYPE

// ---- DUTs/COMPONENTS/PUCK_LOCKER/E_PuckLockerState.TcDUT
{attribute 'qualified_only'}
{attribute 'strict'}
{attribute 'to_string'}
TYPE E_PuckLockerState :
(
	Disabled 					:= 0,
    WaitingForPuck 				:= 10,
    LockingPuck 				:= 20,
    Locked 						:= 30,
	WaitingForNestsEmpty 		:= 35,
    ReleasingPucks 				:= 40,
    UnexpectedPuckRemovalFault 	:= 99
);
END_TYPE

// ---- DUTs/COMPONENTS/PUCK_LOCKER/ST_PuckLocker.TcDUT
TYPE ST_PuckLocker :
STRUCT
	eState                  : E_PuckLockerState;
	
	bNestsEmpty 			: BOOL;
    
	bPuckSensorUp           : BOOL;
    bPuckSensorDown         : BOOL;
    bPuckDetected           : BOOL;
    bPuckSensorMismatch     : BOOL;

    bPinCommandUp           : BOOL;
    bPuckLocked             : BOOL;

    bRemovalAllowed         : BOOL;
    bUnexpectedRemovalFault : BOOL;

    nPucksAllowedToPass     : USINT;
    nPucksToRemove          : USINT;

    bApplyDisposition       : BOOL;
    nRequestedRelease       : USINT;
    nRequestedRemoval       : USINT;

    bDispositionPending     : BOOL;
    bDispositionHandled     : BOOL;

    sMessage                : STRING(255);
END_STRUCT
END_TYPE

// ---- DUTs/COMPONENTS/PUCK_LOCKER/ST_PuckLockerHMI.TcDUT
TYPE ST_PuckLockerHMI :
STRUCT
	eMode                       : E_PuckLockerMode;

    bEnableEmptyPuckBypass      : BOOL;
    bCmdEmptyPuckBypass         : BOOL;
    bCmdAcknowledgeRemovalFault : BOOL;

    bPuckDetected               : BOOL;
    bPuckLocked                 : BOOL;
    bPuckSensorMismatch         : BOOL;

    bUnexpectedRemovalFault     : BOOL;
    bShowUnexpectedRemovalPopup : BOOL;
    bShowEmptyPuckPopup         : BOOL;

    nPucksAllowedToPass         : USINT;
    sMessage                    : STRING(255);
END_STRUCT
END_TYPE

// ---- DUTs/HMI/ST_Animations.TcDUT
TYPE ST_Animations :
STRUCT
	
	abDistanceBoxesGreen							: ARRAY[0..5] OF BOOL;


END_STRUCT
END_TYPE

// ---- DUTs/HMI/ST_StatisticsHMI.TcDUT
TYPE ST_StatisticsHMI :
STRUCT
	
	sName					: STRING;
	nGood					: DINT;
	nBad					: DINT;
	bResetGood				: BOOL;
	bResetBad				: BOOL;	
	nEfficency				: STRING;
	
END_STRUCT
END_TYPE

// ---- DUTs/HMI/ST_StatusBanner.TcDUT
TYPE ST_StatusBanner :
STRUCT
	
	sMachineStatusText					:STRING;
	nMachineStatusTxtCol				:DWORD;
	nMachineStatusColour				:DWORD;
	sBannerTextColor					:STRING;
	sBannerBckColor						:STRING;
	

END_STRUCT
END_TYPE

// ---- DUTs/IO/CAMERA/ST_KeyenceCamera_I_O.TcDUT
TYPE ST_KeyenceCamera_I_O :
STRUCT
	
///////////////////////////////////////////////////////////////INPUTS////////////////////////////////////////////////////////////////////

	bResultReady							AT %I*			: BOOL;	
	bTriggerFail							AT %I*			: BOOL;	
	bError									AT %I*			: BOOL;	
	bAlarm									AT %I*			: BOOL;	
	bBusy									AT %I*			: BOOL;	
	bRun									AT %I*			: BOOL;	
	bReady									AT %I*			: BOOL;	
	bTotalResult							AT %I*			: BOOL;	
	nScore									AT %I*			: UINT;	

///////////////////////////////////////////////////////////////OUTPUTS////////////////////////////////////////////////////////////////////

	bTrigger								AT %Q*			: BOOL;				
	bReset									AT %Q*			: BOOL;	
	bSetTreshold							AT %Q*			: BOOL;	
	bResultReadyAck							AT %Q*			: BOOL;	
	bSettingNo								AT %Q*			: UINT;	
	bSettingVal								AT %Q*			: UDINT;	
	bResetStatistics						AT %Q*			: BOOL;	
	bClearBuffer							AT %Q*			: BOOL;
	
END_STRUCT
END_TYPE

// ---- DUTs/IO/CARDS/ST_EL1918_C.TcDUT
TYPE ST_EL1918_C :
STRUCT
	//--------------------------------------------------------------------------------------------------------
	sTerminalName                                           :   STRING(200):= 'EL1918 | 8-Channel Safety Digital Input';
    //============================================================================================================================	
	// TERMINAL - EL1918 8-Channel Digital Input Terminal 	(Term 5)

	iD3ProcessCylinderRetracted1            AT %I*			: 	BOOL;	// EL1918 channel 1
	iD3ProcessCylinderRetracted2           	AT %I*			: 	BOOL;	// EL1918 channel 2
	iD3ProcessCylinderFeedback        		AT %I*	 		: 	BOOL;	// EL1918 channel 3
	iEL1918_Ch4   							AT %I*	 		: 	BOOL;	// EL1918 channel 4
	iEL1918_Ch5         					AT %I*	 		: 	BOOL;	// EL1918 channel 5 		     			
	iEL1918_Ch6								AT %I*			: 	BOOL;	// EL1918 channel 6
	iEL1918_Ch7              				AT %I*          :   BOOL;   // EL1918 channel 7 
    iEL1918_Ch8          					AT %I*          :   BOOL;   // EL1918 channel 8
 		
	stTerminalInfo											: 	ST_Terminal_Info;

END_STRUCT
END_TYPE

// ---- DUTs/IO/CARDS/ST_EL1918_A.TcDUT
TYPE ST_EL1918_A :
STRUCT
	//--------------------------------------------------------------------------------------------------------
	sTerminalName                                           :   STRING(200):= 'EL1918 | 8-Channel Safety Digital Input';
    //============================================================================================================================	
	// TERMINAL - EL1918 8-Channel Digital Input Terminal (Term 4)	
	iEStopChannel1                			AT %I*			: 	BOOL;	// EL1918 channel 1
	iEStopChannel2                   		AT %I*			: 	BOOL;	// EL1918 channel 2
	iResetButton        					AT %I*	 		: 	BOOL;	// EL1918 channel 3
	iD1MainDoorLocked1   					AT %I*	 		: 	BOOL;	// EL1918 channel 4
	iD1MainDoorLocked2         				AT %I*	 		: 	BOOL;	// EL1918 channel 5 		     			
	iD1MainDoorFB 							AT %I*			: 	BOOL;	// EL1918 channel 6
	iFestoMS6ValveFB               			AT %I*          :   BOOL;   // EL1918 channel 7 
    iFestoMS6DumpValveFB          			AT %I*          :   BOOL;   // EL1918 channel 8
 		
	stTerminalInfo											: 	ST_Terminal_Info;

END_STRUCT
END_TYPE

// ---- DUTs/IO/CARDS/ST_EL1918_B.TcDUT
TYPE ST_EL1918_B :
STRUCT
	//--------------------------------------------------------------------------------------------------------
	sTerminalName                                           :   STRING(200):= 'EL1918 | 8-Channel Safety Digital Input';
    //============================================================================================================================	
	// TERMINAL - EL1918 8-Channel Digital Input Terminal 	(Term 5)

	iRightTouchButtonNC                		AT %I*			: 	BOOL;	// EL1918 channel 1
	iLeftTouchButtonNC                   	AT %I*			: 	BOOL;	// EL1918 channel 2
	iRightTouchButtonNO        				AT %I*	 		: 	BOOL;	// EL1918 channel 3
	iLeftTouchButtonNO   					AT %I*	 		: 	BOOL;	// EL1918 channel 4
	iProcessDoorClosed1         			AT %I*	 		: 	BOOL;	// EL1918 channel 5 		     			
	iProcessDoorClosed2 					AT %I*			: 	BOOL;	// EL1918 channel 6
	iProcessDoorFB               			AT %I*          :   BOOL;   // EL1918 channel 7 
    iEL1918_Ch8          					AT %I*          :   BOOL;   // EL1918 channel 8
 		
	stTerminalInfo											: 	ST_Terminal_Info;

END_STRUCT
END_TYPE

// ---- DUTs/IO/CARDS/ST_EL2904.TcDUT
TYPE ST_EL2904 :
STRUCT
	//--------------------------------------------------------------------------------------------------------
	sTerminalName                                           :   STRING(200):= 'EL2904 | 4-Channel Digital Output';
	//=============================================================================================================
	// TERMINAL - EL2904	4-Channel Digital Output Terminal	 (Term 6)
	qEnableAirSupply_PSR1 					AT %Q*			: 	BOOL;	// EL2904 channel 1
	qResetAirSupply_PSR2					AT %Q* 			: 	BOOL;	// EL2904 channel 2
	qLockMainDoor             				AT %Q*	 		: 	BOOL;	// EL2904 channel 3 			
	qLockProcessCylinder      				AT %Q*	 		: 	BOOL;	// EL2904 channel 4 
	
	stTerminalInfo											: 	ST_Terminal_Info;
	
END_STRUCT
END_TYPE

// ---- DUTs/IO/CARDS/ST_EL6910.TcDUT
TYPE ST_EL6910 :
STRUCT
	
	// TERMINAL - EL6910	TwinSAFE logic	 (Term 3)
	sTerminalName                                           :   STRING(200):= 'EL6910 | TwinSAFE logic';
	stTerminalInfo											: 	ST_Terminal_Info;

END_STRUCT
END_TYPE

// ---- DUTs/IO/CARDS/ST_EL6633.TcDUT
TYPE ST_EL6633 :
STRUCT
	
	// TERMINAL - EL66633	Profinet Protocol	 (Term 12)
	sTerminalName                                           :   STRING(200):= 'EL6633 | Profinet Protocol';
	stTerminalInfo											: 	ST_Terminal_Info;

END_STRUCT
END_TYPE

// ---- DUTs/IO/CARDS/ST_EL9410.TcDUT
TYPE ST_EL9410 :
STRUCT
	
	// TERMINAL - EL9410	E-Bus Power supply	 (Term 7)
	sTerminalName                                           :   STRING(200):= 'EL9410 | E-Bus Power supply';
	stTerminalInfo											: 	ST_Terminal_Info;

END_STRUCT
END_TYPE

// ---- DUTs/IO/CARDS/ST_EL1809.TcDUT
TYPE ST_EL1809 :
STRUCT
	//--------------------------------------------------------------------------------------------------------
	sTerminalName                                           :   STRING(200):= 'EL1809 | 16-Channel Digital Input';
    //============================================================================================================================	
	// TERMINAL - EL1809 16-Channel Digital Input Terminal (Term 8)	
	iStartButoon                			AT %I*			: 	BOOL;	// EL1809 channel 1
	iStopButton                   			AT %I*			: 	BOOL;	// EL1809 channel 2
	iUP_OK        							AT %I*	 		: 	BOOL;	// EL1809 channel 3
	iUS_OK		   							AT %I*	 		: 	BOOL;	// EL1809 channel 4
	iPartPresentNest1         				AT %I*	 		: 	BOOL;	// EL1809 channel 5 		     			
	iPartPresentNest2 						AT %I*			: 	BOOL;	// EL1809 channel 6
	iEL1809_Ch7               				AT %I*          :   BOOL;   // EL1809 channel 7 
    iEL1809_Ch8          					AT %I*          :   BOOL;   // EL1809 channel 8
    iEL1809_Ch9           					AT %I*          :   BOOL;   // EL1809 channel 9
	iProcessCylinderExtended              	AT %I*          :   BOOL;   // EL1809 channel 10
	iRejectSensor              				AT %I*          :   BOOL;   // EL1809 channel 11
	iEL1809_Ch12			              	AT %I*          :   BOOL;   // EL1809 channel 12	   
	iEL1809_Ch13         		   			AT %I*	 		: 	BOOL;	// EL1809 channel 13   
	iEL1809_Ch14       						AT %I*	 		: 	BOOL;	// EL1809 channel 14 
	iPuckSensorUp	(*Renan Added 06/07*)	AT %I*			: 	BOOL;	// EL1809 channel 15  
	iPuckSensorDown	(*Renan Added 06/07*)	AT %I*	 		: 	BOOL;	// EL1809 channel 16  	
	
	stTerminalInfo											: 	ST_Terminal_Info;

END_STRUCT
END_TYPE

// ---- DUTs/IO/CARDS/ST_EL2809_A.TcDUT
TYPE ST_EL2809_A :
STRUCT
	//--------------------------------------------------------------------------------------------------------
	sTerminalName                                           :   STRING(200):= 'EL2809 | 16-Channel Digital Output';
	//=============================================================================================================
	// TERMINAL - EL2809	16-Channel Digital Output Terminal	 (Term 9)
	qResetButtonLED 						AT %Q*			: 	BOOL;	// EL2809 channel 1
	qStartButtonLED							AT %Q* 			: 	BOOL;	// EL2809 channel 2
	qOpenProcessDoor             			AT %Q*	 		: 	BOOL;	// EL2809 channel 3 			
	qCloseProcessDoor      					AT %Q*	 		: 	BOOL;	// EL2809 channel 4 
	qRetractProcessCylinder  				AT %Q*	 		: 	BOOL;	// EL2809 channel 5
	qExtendProcessCylinder	 				AT %Q*	 		: 	BOOL;	// EL2809 channel 6 	
	qPanelLightLED         		    		AT %Q*			: 	BOOL;	// EL2809 channel 7	
	qIndicatorLED1_Red						AT %Q*	 		: 	BOOL;	// EL2809 channel 8	
	qIndicatorLED1_Green                 	AT %Q*          :   BOOL;   // EL2809 channel 9
	qIndicatorLED2_Red             			AT %Q*          :   BOOL;   // EL2809 channel 10   	
	qIndicatorLED2_Green     				AT %Q*	 		: 	BOOL;	// EL2809 channel 11	
	qiEL2809_Ch12   						AT %Q*	 		: 	BOOL;	// EL2809 channel 12 
    qiEL2809_Ch13			        		AT %Q*	 		: 	BOOL;	// EL2809 channel 13 
	qiEL2809_Ch14                 			AT %Q*	 		: 	BOOL;	// EL2809 channel 14 
	qiEL2809_Ch15							AT %Q*	 		: 	BOOL;	// EL2809 channel 15 
    qPuckLockerPinCommand  	        	AT %Q*	 		: 	BOOL;	// EL2809 channel 16
	
	stTerminalInfo											: 	ST_Terminal_Info;
	
END_STRUCT
END_TYPE

// ---- DUTs/IO/LEAK_TESTERS/st_i28General_I_O.TcDUT
TYPE st_i28General_I_O :
STRUCT
	
//OUTPUTS
bOutput1	                   	AT%Q*       : BOOL;
bOutput2	                   	AT%Q*       : BOOL;
bOutput3	                   	AT%Q*       : BOOL;
bOutput4	                   	AT%Q*       : BOOL;
bOutput5	                   	AT%Q*       : BOOL;
bOutput6	                   	AT%Q*       : BOOL;
bOutput7	                   	AT%Q*       : BOOL;
bOutput8	                   	AT%Q*       : BOOL;
bOutput9	                   	AT%Q*       : BOOL;
bOutput10	                   	AT%Q*       : BOOL;
bOutput11	                   	AT%Q*       : BOOL;
bOutput12	                   	AT%Q*       : BOOL;
bOutput13	                   	AT%Q*       : BOOL;
bOutput14	                   	AT%Q*       : BOOL;
bOutput15	                   	AT%Q*       : BOOL;
bOutput16	                   	AT%Q*       : BOOL;

bChangeProgram	                AT%Q*       : BOOL;
bVentHalt	                	AT%Q*       : BOOL;
bReset	                		AT%Q*       : BOOL;
bStop	                		AT%Q*       : BOOL;
bStart	                		AT%Q*       : BOOL;

bSetProgram						AT%Q*       : ARRAY [0..7] OF BOOL;


//i28 inputs
bInput1			               	AT%I*       : BOOL; 
bInput2			               	AT%I*       : BOOL; 
bInput3			               	AT%I*       : BOOL; 
bInput4			               	AT%I*       : BOOL; 
bInput5			               	AT%I*       : BOOL; 
bInput6			               	AT%I*       : BOOL; 
bInput7			               	AT%I*       : BOOL; 
bInput8			               	AT%I*       : BOOL; 
bInput9			               	AT%I*       : BOOL; 
bInput10		               	AT%I*       : BOOL; 
bInput11		               	AT%I*       : BOOL; 
bInput12		               	AT%I*       : BOOL; 
bInput13		               	AT%I*       : BOOL; 
bInput14		               	AT%I*       : BOOL; 
bInput15		               	AT%I*       : BOOL; 
bInput16		               	AT%I*       : BOOL; 

bTestActiveLiveData			   	AT%I*       : BOOL;
bMalfunction	               	AT%I*       : BOOL; 
bProgramReject	               	AT%I*       : BOOL; 
bProgramAccept	               	AT%I*       : BOOL; 
bInstrumentReady               	AT%I*       : BOOL;
nCurrentProgramNumber			AT%I*		: USINT; 




END_STRUCT
END_TYPE

// ---- DUTs/IO/LEAK_TESTERS/st_i28LasResult.TcDUT
TYPE st_i28LasResult :
STRUCT

inUniqueID			               	AT%I*       : UDINT; 
inChannelNumber						AT%I*       : USINT;
inProgramNumber						AT%I*       : USINT;
inTestPort							AT%I*       : USINT;
inPartEvaluation					AT%I*       : USINT;
inTestType							AT%I*       : USINT;
inPrecisionCode						AT%I*       : USINT;

ibTestEvaluation0					AT%I*       : BOOL;
ibTestEvaluation1					AT%I*       : BOOL;
ibTestEvaluation2					AT%I*       : BOOL;
ibTestEvaluation3					AT%I*       : BOOL;


inMeasurement1						AT%I*       : UDINT;
inVariableCode1						AT%I*       : UINT;
inUnitCode1							AT%I*       : USINT;


inMeasurement2						AT%I*       : UDINT;
inVariableCode2						AT%I*       : UINT;
inUnitCode2							AT%I*       : USINT;

//Output Data
sPartEvaluation									: WSTRING;
sTestType										: WSTRING;
sPrecision										: WSTRING;
sTestEvaluation									: WSTRING;
sVariable1										: WSTRING; 
sUnit1											: WSTRING;
sVariable2										: WSTRING; 
sUnit2											: WSTRING;

//Info
sDate											: STRING;
sTime											: STRING;









END_STRUCT
END_TYPE

// ---- DUTs/IO/LEAK_TESTERS/st_i28LiveMeasurement.TcDUT
TYPE st_i28LiveMeasurement :
STRUCT

inUniqueID			               	AT%I*       : UDINT; 
inCurrentProgramNumber				AT%I*       : UINT;
inSegmentCode						AT%I*       : USINT;

inMeasurement1						AT%I*       : UDINT;//TIME
inVariableCode1						AT%I*       : UINT;
inUnitCode1							AT%I*       : USINT;
inPrecisionCode1					AT%I*       : USINT;

inMeasurement2						AT%I*       : UDINT;//PRESSURE
inVariableCode2						AT%I*       : UINT;
inUnitCode2							AT%I*       : USINT;
inPrecisionCode2					AT%I*       : USINT;

inMeasurement3						AT%I*       : UDINT;//PRESSURE LOSS/RATE
inVariableCode3						AT%I*       : UINT;
inUnitCode3							AT%I*       : USINT;
inPrecisionCode3					AT%I*       : USINT;

inMeasurement4						AT%I*       : UDINT;//FLOW/LEAK
inVariableCode4						AT%I*       : UINT;
inUnitCode4							AT%I*       : USINT;
inPrecisionCode4					AT%I*       : USINT;



//Output Data
sSegmentCode									:WSTRING;


sVariable1										:WSTRING;
sUnit1											:WSTRING;
sPrecision1										:WSTRING;


sVariable2										:WSTRING;
sUnit2											:WSTRING;
sPrecision2										:WSTRING;


sVariable3										:WSTRING;
sUnit3											:WSTRING;
sPrecision3										:WSTRING;


sVariable4										:WSTRING;
sUnit4											:WSTRING;
sPrecision4										:WSTRING;



END_STRUCT
END_TYPE

// ---- DUTs/IO/PROBES/ST_ProbesSet.TcDUT
TYPE ST_ProbesSet :
STRUCT
	
	abProbeError							AT %I*			: ARRAY[1..4] OF BOOL;
	anRawMeasurement						AT %I*			: ARRAY[1..4] OF DINT;
	anScaledRawMeasurement									: ARRAY[1..4] OF REAL;
	
END_STRUCT
END_TYPE

// ---- DUTs/IO/PROBES/ST_Probes_I_O.TcDUT
TYPE ST_Probes_I_O :
STRUCT
	
	bGeneralError					AT %I*					: BOOL;
	stProbesSet												: ARRAY [1..2] OF ST_ProbesSet;
	abPresetProbe					AT %Q*					: DINT;
	
	stTerminalInfo											: 	ST_Terminal_Info;
	
END_STRUCT
END_TYPE

// ---- DUTs/MASTER/E_MachineState.TcDUT
{attribute 'qualified_only'}
{attribute 'strict'}
TYPE E_MachineState :
(
	SYSTEM_POWER_UP			,
	STOPPED					,
	SYSTEM_INITIALISING		,
	SYSTEM_READY_TO_START	,
	SYSTEM_AUTO_CYCLE		,
	STOPPING				,
	MANUAL_MODE				,
	FAULT					,
	SAFETY
);
END_TYPE

// ---- DUTs/MASTER/log_CSV/ST_UserLog.TcDUT
TYPE ST_UserLog :
STRUCT
	
	sUser				: STRING;
	sGroup				: STRING;
	sDate				: STRING;
	sTime				: STRING;
	
END_STRUCT
END_TYPE

// ---- DUTs/MASTER/PROCESS CYCLES/E_General_ProcessCycle.TcDUT
{attribute 'qualified_only'}
{attribute 'strict'}
TYPE E_General_ProcessCycle :
(
	
IDLE								,
PROCESS_FLAGS_DEFINITIONS			,
CLOSE_PROCESS_DOOR					,
WAIT_CLOSE_PROCESS_DOOR				,
OPEN_PROCESS_DOOR					,
WAIT_OPEN_PROCESS_DOOR				,
PRE_RETRACT_PROCESS_CYLINDER		,	//Renan added - Buglist n13 - 08Jul26
WAIT_PRE_RETRACT_PROCESS_CYLINDER	, 	//Renan added - Buglist n13 - 08Jul26
EXTEND_PROCESS_CYLINDER				,
WAIT_EXTEND_PROCESS_CYLINDER		,
RETRACT_PROCESS_CYLINDER			,
WAIT_RETRACT_PROCESS_CYLINDER		,
CAMERA_INSPECTION					,
WAIT_CAMERA							,
LEAK_TESTS							,
WAIT_LEAK_TEST						,
LEAK_TESTS_HEIGHT_TEST				,
WAIT_LEAK_TEST_HEIGHT_TEST			,
HEIGHT_TEST							,
WAIT_HEIGHT_TEST					,
WAIT_TO_SAVE_DATA					,
WAIT_RESULTS						,
RESULTS								,
SAVE_DATA							,
SAVE_DATA2							,
CSV_NEST1							,
CSV_NEST2							,
REJECT_CHUTE_FULL					,
WAIT_REJECT_PART					,
PUCK_DEFINITION						,
NEST_CLEARING						,

RESET_ALL_CMD						

);
END_TYPE

// ---- DUTs/MASTER/ST_ButtonsLamps.TcDUT
TYPE ST_ButtonsLamps :
STRUCT
		
	bStartButtonRisingEdge			: 	BOOL;
	bStartButtonFallingEdge			:	BOOL;
	bResetButtonRisingEdge			: 	BOOL;
	bResetButtonFallingEdge			: 	BOOL;
	bStopButtonRisingEdge			:	BOOL;
	bStopButtonFallingEdge			:	BOOL;
	
	
	
END_STRUCT
END_TYPE

// ---- DUTs/MASTER/ST_MACHINE.TcDUT
TYPE ST_MACHINE :
STRUCT
	
	sName						: STRING;
	
	bMachine					: ARRAY [1..3] OF BOOL;
		
	bHeightTest 				: BOOL;
	bVisionTest					: BOOL;
	bLeakTest					: BOOL;
	bPuckLocker				: BOOL; //Renan Added 10Jul26 - Puck Locker

END_STRUCT
END_TYPE

// ---- DUTs/MASTER/ST_MachineStatus.TcDUT
TYPE ST_MachineStatus :
STRUCT
	////////////////////////////:
	eMachineState				:E_MachineState;
	
	// Status Flags:
	bSystemPowerUp 				:BOOL;
	bStopped 					:BOOL;
	bInitialising 				:BOOL;
	bReadyToStart 				:BOOL;
	bAutoCycle 					:BOOL;
	bStopping					:BOOL;
	bFault 						:BOOL;
	bManualMode					:BOOL;
	bSafety						:BOOL;

END_STRUCT
END_TYPE

// ---- DUTs/MASTER/ST_MasterCTRL.TcDUT
TYPE ST_MasterCTRL :
STRUCT
	

	// Request Flags
	bManualModeRequest					:BOOL;
	
	bCycleStopRequest					:BOOL;
	
	bNoFault							:BOOL;
	
	// Feedback Flags
	bAllStationsReady					:BOOL;
	bAllStationsStopped					:BOOL;
	
	bPowerUpTimerComplete				:BOOL;

	
//-------------------------------------------------------------------------------oldschoo1
		
END_STRUCT
END_TYPE

// ---- DUTs/MASTER/ST_Puls.TcDUT
TYPE ST_Puls :
STRUCT
	
	bFlash1Hz						: BOOL;
	bFlash2Hz						: BOOL;
	bFlash4Hz				   		: BOOL;
	bFlash10Hz						: BOOL;
	bFlash10BHz        		  		: BOOL;
	bFlash100Hz      	      		: BOOL;
	bFlashScale       	      		: BOOL;
	bFlashScale4       		  		: BOOL;
	bFlashScale5        	  		: BOOL;
	bFlash5sec                      : BOOL;
	
END_STRUCT
END_TYPE

// ---- DUTs/COMPONENTS/CAMERA/E_Camera_State.TcDUT
{attribute 'qualified_only'}
{attribute 'strict'}
TYPE E_Camera_State :
(
	//GENERIC
	ABORTED				,
	RESET_ERROR			,
	READY				,
	RESET_CMD			,
	//MANUAL_MODE			:=50, /manual mode not needed.
	ERROR				,
	//SPECIFIC FOR EVERY STATION
	HOMING				,
	
	TAKING_PICTURE_CAP	,
	TAKING_PICTURE_FPB	,
	COMPARING_RESULTS	,
	DONE				,
	RESULTS_CAP			,
	RESULTS_FPB				
);
END_TYPE

// ---- DUTs/COMPONENTS/HEIGHT TEST/E_HeightTest_State.TcDUT
{attribute 'qualified_only'}
{attribute 'strict'}
TYPE E_HeightTest_State :
(
	//GENERIC
	ABORTED				,
	READY				,
	//MANUAL_MODE			:=50, /manual mode not needed.
	ERROR				,
	//SPECIFIC FOR EVERY STATION
	MEASURE				,
	WAIT_MEASUREMENT	,
	DONE				,
	RESULTS				,
	RESET				,
	MANUAL_MODE
);
END_TYPE

// ---- DUTs/COMPONENTS/MAIN CYLINDER/E_ProcessCylinder_State.TcDUT
{attribute 'qualified_only'}
{attribute 'strict'}
TYPE E_ProcessCylinder_State :
(
		//GENERIC
	ABORTED				,
	HOMING				,
	READY				,
	MANUAL_MODE			,
	STOPPING			,
	//SPECIFIC FOR EVERY STATION
	EXTEND,
	RETRACT,
	DONE				,
	RESET				
);
END_TYPE

// ---- DUTs/ST_TwinSAFE.TcDUT
TYPE ST_TwinSAFE :
STRUCT
	
///////////////////////////////////////////////////////////////////////////Safety OUTPUTS///////////////////////////////////////////////////////////////////////////////////////
		
	iAirPressureMaxValue					AT %Q*			: 	UINT;
	iAirPressureMinValue					AT %Q*			: 	UINT;
	iAirSupplyMeasurement					AT %Q*			: 	UINT;
	iMachineStopped							AT %Q*			: 	BOOL;	
	iProcessDoorClosing              		AT %Q*			: 	BOOL;		
	iProcessDoorClosedCondition				AT %Q*			: 	BOOL;
	iSafetyErrorAcknowledge					AT %Q*			: 	BOOL;
	iRunSafety								AT %Q*			: 	BOOL;
	iInitSafety								AT %Q*			: 	BOOL;
	iMachineHoming_Manual					AT %Q*			: 	BOOL;
	iPuckError								AT %Q*			: 	BOOL; //Renan Added 10Jul26 - Puck Locker
	
///////////////////////////////////////////////////////////////////////////Safety Inputs///////////////////////////////////////////////////////////////////////////////////////	

	qAirErrorSignal							AT %I*			: 	BOOL;	
	qAirPressureAbove						AT %I*			: 	BOOL;	
	qAirPressureBelow						AT %I*			: 	BOOL;
	qAirPressureOK							AT %I*			: 	BOOL;
	qMainDoorOpenned						AT %I*			: 	BOOL;	
	qE_StopPressed							AT %I*			: 	BOOL;	
	qMainDoorUnsafe							AT %I*			: 	BOOL;	
	qProcessCylinderUnsafe					AT %I*			: 	BOOL;
	qProcessCylinderRetracted				AT %I*			: 	BOOL;
	qProcessDoorUnSafe						AT %I*			: 	BOOL;	
	qSafetyOk								AT %I*			: 	BOOL;
	qSystemSafe								AT %I*			: 	BOOL;
	qTwoHandsUnsafe							AT %I*			: 	BOOL;
	qFBError								AT %I*			: 	BOOL;
	qOtherError								AT %I*			: 	BOOL;
	qComError								AT %I*			: 	BOOL;
	qTwoHandsSafe							AT %I*			: 	BOOL;

END_STRUCT
END_TYPE

// ---- DUTs/USER_ALARMS_EVENTS/EVENTS/ST_ActiveEvents.TcDUT
TYPE ST_ActiveEvents :
STRUCT
	
	sEventTex									: STRING(255);
	sType										: STRING(255);
	sSolution									: STRING(255);
	abType										: DINT;					//1:Alarm
																		//2:Alert
																		//3:Message

END_STRUCT
END_TYPE

// ---- DUTs/USER_ALARMS_EVENTS/EVENTS/ST_EventsAssigment.TcDUT
TYPE ST_EventsAssigment :
STRUCT
	
	sEventText							: STRING(255);
	sSolution							: STRING(255);
	
END_STRUCT
END_TYPE

// ---- DUTs/USER_ALARMS_EVENTS/EVENTS/ST_EventsAssigmentGeneral.TcDUT
TYPE ST_EventsAssigmentGeneral :
STRUCT
	
	astFaultEvents						: ARRAY [1..100] OF ST_EventsAssigment;
	astCycleStopRequestEvents			: ARRAY [1..100] OF ST_EventsAssigment;
	astMessage							: ARRAY [1..100] OF ST_EventsAssigment;
	
	
END_STRUCT
END_TYPE

// ---- DUTs/USER_ALARMS_EVENTS/EVENTS/ST_EVENT.TcDUT
TYPE ST_EVENT :
STRUCT
	
	bFault								: BOOL;
	bCycleStopRequest					: BOOL;
	bMessage							: BOOL;
	
	bAssignedID							: DINT;
	
	bEventFlag							: BOOL;
	bEventTimer							: TON;
	bEventText							: STRING(255);
	bEventTextHMI						: STRING(255);
	sSolution							: STRING(255);
	bActive								: BOOL;

END_STRUCT
END_TYPE

// ---- DUTs/USER_ALARMS_EVENTS/EVENTS/ST_StationEvents.TcDUT
TYPE ST_StationEvents :
STRUCT
	
	aEvents								: ARRAY [0..100] OF ST_EVENT;	
	
	bFault								: BOOL;
	bCycleStopRequest					: BOOL;
	
			
END_STRUCT
END_TYPE

// ---- DUTs/USER_ALARMS_EVENTS/ST_UserLogHMI.TcDUT
TYPE ST_UserLogHMI :
STRUCT
	UserLog					: T_MaxSTring;
	UserLogTime				: STRING;
	UserLogDate				: STRING;
END_STRUCT
END_TYPE

// ---- GVLs/GVL_HMI.TcGVL
VAR_GLOBAL
////////////////////////////////////////:	///////////////////////////////////////////////////
/////////////////////////////////////////////////////////////////////////////////////GENERIC/////////////////////////////////////////////////////////////////////////////////////

	stHMI_IO							: ST_HMI_IO;
	bQuitHMI							: BOOL;
	bShutDown							: BOOL;
	stStatusBanner						: ST_StatusBanner;
	nPopUp								: DINT;
	
	bPartPresent						: ARRAY [0..1] OF BOOL;
	stStatisticsWH						: ARRAY [0..5] OF ST_StatisticsHMI;
	stStatisticsLT						: ARRAY [0..3] OF ST_StatisticsHMI;
	
	bRejectPartDialog					: ARRAY [0..2] OF BOOL;
	bOpenRejectDialog					: BOOL;
	anCameraScore						: ARRAY [1..4] OF STRING;
	bLightsOnOff						: BOOL;
	
	bHMIAlive							: BOOL;
	tonHMIAliveOn						: TON;
	tonHMIAliveOff						: TON;
	bOutHMI								: BOOL;
	bEmptyRejectChute					: BOOL;
	bEmptyRejectChuteAcknowledge		: BOOL;
	
/////////////////////////////////////////////////////////////////////////////////////SYSTEM INFO/////////////////////////////////////////////////////////////////////////////////////

	sSoftwareVersion					: STRING := ' 1.0 ';
	sSoftwareDate						: STRING := '23/04/2026';
	sTC3Version							: STRING := ' v3.1.4026.22, Runtime v3.1.4026.22 ';
	sHMIVersion							: STRING := ' 14.13';
	sSystemName							: STRING ;
	sProjectID							: STRING := ' TE 11108' ;
	sAplication                     	: STRING ;
	sHMIServer                			: STRING := ' 14.13 ';
	
/////////////////////////////////////////////////////////////////////////////////////MANUAL/////////////////////////////////////////////////////////////////////////////////////

	bEnableManual						: BOOL;
	nMainRegion							: DINT;
	bManualModeOffFlag					: BOOL;
	bManualScreen						: BOOL;
	tonManualMode						: TON;
	bEnableSettings						: BOOL;
	bOnlyHeightTestBypass				: BOOL;

	
	
	stAnimations						: ST_Animations;
	nMachineDefinitionIndex2			: INT;
	bMachineDefinitionSet1				: BOOL;
	rMachineDefinitionSet2				: R_TRIG;
	fMachineDefinitionSet2				: F_TRIG;
	
	bProcessCylinder_Up					: BOOL;
	bProcessCylinder_Up2				: BOOL;
	bProcessCylinder_Down2				: BOOL;
	
	bProcessDoor_Up						: BOOL;
	bProcessDoor_Down					: BOOL;
	
	bLeaktester1_Start					: BOOL;
	bLeaktester2_Start					: BOOL;
	bLeaktester1_Stop					: BOOL;
	bLeaktester2_Stop					: BOOL;
	bLeaktester1_Reset					: BOOL;
	bLeaktester2_Reset					: BOOL;
	bCameraResetStatistics				: ARRAY[1..4] OF BOOL;
	bCameraSettingNo					: ARRAY[1..4] OF UINT;
	bCameraSettingVal					: ARRAY[1..4] OF UDINT;
	bCameraSetTreshold					: ARRAY[1..4] OF BOOL;
	bCameraTrigger						: ARRAY[1..4] OF BOOL;
	
	bProcessCylinderDownEnable			: BOOL;
	
	//Probes
	bSetTolerances						: BOOL;
	abPresetProbe						: ARRAY [1..8] OF BOOL;
	bSetCalibrationBlock1				: BOOL;
	bSetCalibrationBlock2				: BOOL;
	bEnableSetCablibrationBlock1		: BOOL;
	bEnableSetCablibrationBlock2		: BOOL;
	bSetDistances						: BOOL;
	(*Renan Added - 30Jun26 - Getting offset from HMI*)
	bSetProbeOffsetNest1				: BOOL;
	(*/Renan Added - 30Jun26 - Getting offset from HMI*)

	(*Renan Added - 06Jul26 - Getting offset from HMI*)
	//Puck Locker
	stPuckLocker 						: ST_PuckLockerHMI;
	(*\Renan Added - 06Jul26 - Getting offset from HMI*)
	
END_VAR

VAR_GLOBAL PERSISTENT
	
	stTimers							: ST_Timers;
	stStatisticsHMI						: ARRAY [0..7] OF ST_StatisticsHMI;	//0: Nest1
																	//1: Nest2
																	//2: Leak Tester 1
																	//3: Leak Tester 2
																	//4: Height Test 1
																	//5: Height Test 2
																	//6: Camera set 1
																	//7: camera set 2
														
	/////////////////////////////////////////////////////////////////////////////////////SETTINGS/////////////////////////////////////////////////////////////////////////////////////	
	(*Renan Added - 30Jun26 - Getting offset from HMI*)
	anNestOffsetByProbe1         		: ARRAY [1..4] OF REAL;
    anNestOffsetByProbe2         		: ARRAY [1..4] OF REAL;
	(*/Renan Added - 30Jun26 - Getting offset from HMI*)

	(*Renan Added - 06Jul26 - Getting offset from HMI*)
	ePuckLockerMode : E_PuckLockerMode := E_PuckLockerMode.Disabled; //Puck locker state
	bPuckLockerGateEnable 				: BOOL := TRUE;
	bPuckLockerSkipEnable 				: BOOL := FALSE;
	(*\Renan Added - 06Jul26 - Getting offset from HMI*)
	
	//TwinSAFE
	
	nAirPressureMaxValue				: UINT;	
	nAirPressureMinValue				: UINT;	
	abMachineDefinition					: ARRAY[1..5] OF  BOOL;
	stTableCycleDataNest1				: ARRAY[0..2000] OF ST_TableCycleData;
	stTableCycleDataNest2				: ARRAY[0..2000] OF ST_TableCycleData;
	
	bNest1Flag							: BOOL;
	bNest2Flag							: BOOL;
	
	nAmountToEmptyRejectChute			: WORD			:= 20;


	
END_VAR

// ---- GVLs/GVL_IO.TcGVL
VAR_GLOBAL
	
	

	dw_T01_EK1100                                                		: ST_K1100;//EtherCAT Coupler 
	dw_T02_EL6070                                           			: ST_EL6070;//EtherCAT Terminal, license key FOR TwinCAT 3.1 	
	dw_T03_EL6910														: st_EL6910;//TwinSAFE logic
	dw_T04_EL1918														: st_EL1918_A;//EL1918 8 Channel Safety Digital Input
	dw_T05_EL1918														: st_EL1918_B;//EL1918 8 Channel Safety Digital Input
	dw_T06_EL2904														: st_EL2904;//EL2904 4 Channel Safety Digital Output
	dw_T07_EL9410														: st_EL9410;//E-Bus Power supply
	dw_T08_EL1809														: st_EL1809;// 16 Channel Digital Input ( 24VDC )
	dw_T09_EL2809														: st_EL2809_A;// 16 Channel Digital Output ( 24VDC ) 	
	dw_T10_EL3058                                                		: st_EL3058;// 4 Channel Analog Input
	dw_T11_EL1918														: st_EL1918_C;//EL1918 8 Channel Safety Digital Input
	dw_T12_EL6633                                                		: ST_EL6633; // Profinet Protocol
	
	stTwinSAFE															: ST_TwinSAFE;
	
	LeakTester1_IO														: ST_General_LeakTester_I_O;
	LeakTester2_IO														: ST_General_LeakTester_I_O;
	
	Camera1_IO															: ST_KeyenceCamera_I_O;
	Camera2_IO															: ST_KeyenceCamera_I_O;
	Camera3_IO															: ST_KeyenceCamera_I_O;
	Camera4_IO															: ST_KeyenceCamera_I_O;
	
	Probes																: ST_Probes_I_O;

	dw_T06_EL2904_Reading												: ST_SafeOutputsReading;

END_VAR

// ---- GVLs/GVL_Master.TcGVL
VAR_GLOBAL
////////////////////////////////////////:	///////////////////////////////////////////////////
/////////////////////////////////////////////////////////////////////////////////////GENERIC/////////////////////////////////////////////////////////////////////////////////////

	// PowerUP 
	tonSystemPowerUP				:TON;
	tSystemPowerUP_Time				:TIME								:=T#3S;
	bSystemPoweringUP				:BOOL								:=TRUE; //Global System PowerUP Flag
	
	fbSystemShutDown     	        : NT_Shutdown;
	stButtonsLamps					: ST_ButtonsLamps;
	rtrigButton             		: ARRAY[1..3] OF Tc2_Standard.R_TRIG;
	ftrigButton             		: ARRAY[1..3] OF Tc2_Standard.F_TRIG; 
	stPuls							: ST_Puls;		

	stCycleDataNest1				: ST_CycleData;
	stCycleDataNest2				: ST_CycleData;
	
	bWriteNest1						: BOOL;
	bWriteNest2						: BOOL;
	bCSVDone						: BOOL;
	bCSVReady						: BOOL;
	bAutocycleIDLE					: BOOL;
	bDoorOpenedFlag					: BOOL;
	
	bRejectPartFault				: BOOL;
	bRejectPartOutTime				: BOOL;
	bCSVError						: BOOL;
	
	NetAmsIdLocal        	       	: T_AmsNetId;// := '172.18.236.164.1.1'; // AMS-ID for com port setup 
	bReadAMSNetID					: BOOL;
	fbGetLocalAMSNetID				: FB_GetLocalAmsNetId;
	
	fbGetDeviceNetId				: IOF_GetDeviceNetId;
	NetAmsIdDevice					: T_AmsNetId;
	
	bOpenDoorCycleFault				: BOOL;	
	bProcessDoorClosed				: BOOL;
	
	
	
/////////////////////////////////////////////////////////////////////////////////////Event Log/////////////////////////////////////////////////////////////////////////////////////
	
	stStationEvents				: ARRAY[0..4] OF  ST_StationEvents;//0: GENERAL
																	//1: Leak Test
																	//1: Height Test
																	//3: Vision Inspection
																	//4: Cylinders
	astActiveEvents				: ARRAY [0..50] OF ST_ActiveEvents;
	stEventsAssigment			: ST_EventsAssigmentGeneral;
	bMachineMessages			: BOOL;
	sMachineMessage				: STRING;

/////////////////////////////////////////////////////////////////////////////////////MACHINE CONTROL////////////////////////////////////////////////////////////////////////////
	
	stMachineStatus					: ST_MachineStatus;	
	stMasterCtrl					: ST_MasterCTRL;
	bStatisticsTest					: ARRAY[0..6] OF  BOOL;
	
	
////////////////////////////////////////////////////////////////////////////////////SYSTEM////////////////////////////////////////////////////////////////////////////
	stSystemTime				: TIMESTRUCT;
	sSystemTime					: STRING(255);
	sSystemDate					: STRING(255);
	
	bResetTest					: BOOL;
	bTestFlag					: ARRAY[0..10] OF BOOL;

////////////////////////////////////////////////////////////////////////////////////SAFETY////////////////////////////////////////////////////////////////////////////

	bDoorClosingFlag				: BOOL;
	bDoorClosingInitFlag			: BOOL;
	bDoorOpeningFlag				: BOOL;
	bProcessDoorClosedConditionFlag	: BOOL;
	tonSafety						: TON;
	bProcessCylinderSafetyPosition	: BOOL;
	bProcessDoorUpInitialising		: BOOL;
	
END_VAR
VAR_GLOBAL PERSISTENT
	
	stMACHINE						: ST_MACHINE;	//THIS STRUCTURE WILL DEFINDE THE PROCESS IN AUTO CYCLE DEPENDING OF WHAT MACHINE YOU ARE WORKING WITH
													//THE bMachine boolean array will define the machine			//1. LT-WH-VC LEAK TEST: FLUID PATH, HEIGHT TEST: FPB WELDING, VISION CHECK: EWIS FOAM
																													//2. WH: HEIGHT TEST: FPB WELDING
																													//3. LT: LEAK TEST: RESERVOIR 
																													



END_VAR

// ---- GVLs/GVL_Stations.TcGVL
VAR_GLOBAL
	
	
	stCamera								: ST_Camera;
	stLeakTesters							: ST_LeakTester;	
	stHeightTests							: ST_HeightTest;
	stProcessCylinder						: ST_ProcessCylinder;
	stProcessDoor							: ST_ProcessDoor;
	stPuckLocker 							: ST_PuckLocker;
	

END_VAR

// ---- POUs/A_MASTER/A_1_PRG_Main_Master.TcPOU
PROGRAM A_1_PRG_Main_Master
VAR
	
	
	fbStringFormatter       				: Tc2_Utilities.FB_FormatString;
	fbEventsManager							: FB_EventsManager;
	bResetEvents							: BOOL;
	
	ntShutdown								: TC2_Utilities.NT_Shutdown;
	closeChrome 							: NT_StartProcess;
	bCloseChromeBusy						: BOOL;
	tonCloseChromeBusy						: TON;
	//fbUserLog								: FB_UserLog;
	
	
	nFindAdm								: INT;
	nFindEng								: INT;
	nFindOpe								: INT;
	sUserGroupName							: STRING (255);
	sAdmGroup								: STRING (255)							:= 'Administrator';
	sEngGroup								: STRING (255)							:= 'Engineer';
	sOpeGroup								: STRING (255)							:= 'Operator';
	
	rEfficency								: STRING(510);
	
	fbSystemTime							: NT_GetTime;
	
	fbScaleAirSupply						: FB_Scale;
	
	fMessageReset							: F_TRIG;
	j										: DINT;
	i										: DINT;
	b										: DINT; //index quit HMI
	
	rGoodStatistics							: ARRAY [0..1] OF R_TRIG;
	rBadStatistics							: ARRAY [0..1] OF R_TRIG;
	
	cuRejectCounter							: CTU;


				
END_VAR

/////////////////////////////////////////////////////////////////////////////////////GENERAL/////////////////////////////////////////////////////////////////////////////////////
A_3_PRG_FaultHandling();
b_ACT_UserLogout();
a_ACT_ButtonsLamps();
d_ACT_ShutdownAndQuit();
f_ACT_TerminalInfo();
g_ACT_Manual();
h_ACT_Statistics();
i_ACT_TwinSAFE();
j_ACT_MachineDefinition();

C_1_PRG_MainHMI();
//D_1_1_PROG_Write_Data_To_CSV();
//D_2_1_PROG_Write_Data_To_CSV();

PRG_Puls();

// System PowerUP CTRL
tonSystemPowerUP(IN:=bSystemPoweringUP, PT:=tSystemPowerUP_Time);
IF tonSystemPowerUP.Q THEN 
bSystemPoweringUP:=FALSE;
END_IF

/////////////////////////////////////////////////////////////////////////////////////STATIONS/////////////////////////////////////////////////////////////////////////////////////

IF stMACHINE.bHeightTest  THEN
	
	B_2_1_PRG_Master_Height_Test();

END_IF

IF stMACHINE.bLeakTest  THEN
	
	B_1_1_PRG_Master_Leak_Test();

END_IF

IF stMACHINE.bVisionTest THEN
	
	B_3_1_PRG_Master_Camera();

END_IF

B_4_1_PRG_Master_ProcessCylinder();
B_4_2_PRG_Master_ProcessDoor();

/////////////////////////////////////////////////////////////////////////////////////PROCESS/////////////////////////////////////////////////////////////////////////////////////

A_2_PRG_MachineCtrl();
B_5_1_PRG_PuckLocker(); (* Renan Added 06Jul26 - Puck Locker program *)



/////////////////////////////////////////////////////////////////////////////////////EVENT LOG/////////////////////////////////////////////////////////////////////////////////////

fbEventsManager	(			//INPUTS
							bPulse 							:= stPuls.bFlash10Hz, 
							bResetFaults 					:= dw_T04_EL1918.iResetButton, 
							stStationEvents 				:= stStationEvents,
							sSystemTime						:= sSystemTime,
							sSystemDate						:= sSystemDate,
 							stEventsAssigment				:= stEventsAssigment,
							bDataWritedInCSV				:= ,
							nArraySize						:= 4,
							bMachineMessage					:= sMachineMessage,
							
							//OUTPUTS
							astActiveEvents 				=> astActiveEvents,
							astEventsHistory				=> astEventsHistory,
							);



////////////////////////////////////////////////////////////////////////////////////SYSTEM DATE & TIME/////////////////////////////////////////////////////////////////////////////////////

fbSystemTime( START := stPuls.bFlash10Hz, TIMESTR => stSystemTime);
	

sSystemTime					:= 	CONCAT( STR1 := WORD_TO_STRING(stSystemTime.wHour), STR2 := CONCAT( STR1 := ':', STR2 := 
								CONCAT( STR1 := WORD_TO_STRING(stSystemTime.wMinute), STR2 := 
								CONCAT(STR1 := ':', STR2 := WORD_TO_STRING(stSystemTime.wSecond)))));
								
sSystemDate					:= 	CONCAT( STR1 := WORD_TO_STRING(stSystemTime.wDay), STR2 := 
								CONCAT(STR1 := '_', STR2 := CONCAT(STR1 := WORD_TO_STRING(stSystemTime.wMonth), STR2 := 
								CONCAT(STR1 := '_', STR2 := WORD_TO_STRING(stSystemTime.wYear)))));


stCycleDataNest1.nNest		:= 1;
stCycleDataNest2.nNest		:= 2;

////////////////////////////////////////////////////////////////////////////////////CSV////////////////////////////////////////////////////////////////////////////	

	

D_1_PRG_CycleDataCSV( 	stCycleDataNest1 	:= stCycleDataNest1,
						stCycleDataNest2 	:= stCycleDataNest2,
						bWriteNest1			:= bWriteNest1,
						bWriteNest2			:= bWriteNest2,
						bCSVDone			=> bCSVDone,
						bReady				=> bCSVReady);
	
fbGetLocalAMSNetID(
					bExecute	:= bReadAMSNetID,
					AddrString => NetAmsIdLocal);	

fbGetDeviceNetId(	START		:= 	bReadAMSNetID,
					DEVICEID	:= 3,
					DeviceNetId	=> 	NetAmsIdDevice);

ACTION a_ACT_ButtonsLamps:
//===================================================================
stButtonsLamps.bStartButtonFallingEdge 		:= ftrigButton[1].Q ;
stButtonsLamps.bStartButtonRisingEdge 		:= rtrigButton[1].Q ;
stButtonsLamps.bStopButtonFallingEdge 		:= ftrigButton[2].Q ; 
stButtonsLamps.bStopButtonRisingEdge 		:= rtrigButton[2].Q ;  
stButtonsLamps.bResetButtonFallingEdge 		:= ftrigButton[3].Q ;
stButtonsLamps.bResetButtonRisingEdge 		:= rtrigButton[3].Q ;



ftrigButton[1](CLK 							:= dw_T08_EL1809.iStartButoon);
rtrigButton[1](CLK							:= dw_T08_EL1809.iStartButoon);
ftrigButton[2](CLK							:= NOT dw_T08_EL1809.iStopButton);
rtrigButton[2](CLK							:= NOT dw_T08_EL1809.iStopButton);
ftrigButton[3](CLK							:= dw_T04_EL1918.iResetButton);
rtrigButton[3](CLK							:= dw_T04_EL1918.iResetButton);

dw_T09_EL2809.qResetButtonLED				:= (stMachineStatus.bFault AND stPuls.bFlash1Hz) OR (stMachineStatus.bStopped AND stPuls.bFlash2Hz) OR stMachineStatus.bManualMode;
dw_T09_EL2809.qStartButtonLED				:= (stMachineStatus.bReadyToStart AND stPuls.bFlash1Hz) OR stMachineStatus.bAutoCycle OR stMachineStatus.bManualMode;
END_ACTION

ACTION b_ACT_UserLogout:
tonHMIAliveOn(IN := bHMIAlive, PT:= T#2S);

tonHMIAliveOff(IN := NOT bHMIAlive, PT:= T#2S);

bOutHMI := tonHMIAliveOn.Q OR tonHMIAliveOff.Q;
END_ACTION

ACTION d_ACT_ShutdownAndQuit:
tonCloseChromeBusy( IN := bQuitHmi, PT := T#5S);
IF  tonCloseChromeBusy.Q THEN
	
	bQuitHmi			:= FALSE;

END_IF

closeChrome(
    NetId := NetAmsIdLocal,
    PathStr := 'C:\Windows\System32\mshta vbscript:Execute("CreateObject(""WScript.Shell"").Run ""powershell -c',
    DirName := 'C:\Windows\System32\WindowsPowerShell\v1.0',
    ComndLine := 'taskkill /F /IM msedge.exe /T"", 0: window.close")',
    Start := bQuitHmi,
    TmOut := DEFAULT_ADS_TIMEOUT,
	BUSY => bCloseChromeBusy
);


ntShutdown(NETID := NetAmsIdLocal, DELAY := 5, START := bShutDown);

IF dw_T08_EL1809.iStartButoon THEN
	IF ftrigButton[2].Q THEN
		b:= b+1;
	END_IF
	IF b>=3 THEN;
		bQuitHmi:=TRUE;
	END_IF
ELSE
	b:=0;
END_IF
END_ACTION

ACTION f_ACT_TerminalInfo:
dw_T01_EK1100.stTerminalInfo.fbTerminalInfo( 	nTerminalState						:= dw_T01_EK1100.stTerminalInfo.nTerminal_State,
												sTerminalState						=> dw_T01_EK1100.stTerminalInfo.sTerminalInfo,
												bTerminalOperational				=> dw_T01_EK1100.stTerminalInfo.bTerminalOperational);
									
dw_T02_EL6070.stTerminalInfo.fbTerminalInfo( 	nTerminalState						:= dw_T02_EL6070.stTerminalInfo.nTerminal_State,
												sTerminalState						=> dw_T02_EL6070.stTerminalInfo.sTerminalInfo,
												bTerminalOperational				=> dw_T02_EL6070.stTerminalInfo.bTerminalOperational);

dw_T03_EL6910.stTerminalInfo.fbTerminalInfo( 	nTerminalState						:= dw_T03_EL6910.stTerminalInfo.nTerminal_State,
												sTerminalState						=> dw_T03_EL6910.stTerminalInfo.sTerminalInfo,
												bTerminalOperational				=> dw_T03_EL6910.stTerminalInfo.bTerminalOperational);
												
dw_T04_EL1918.stTerminalInfo.fbTerminalInfo(	nTerminalState						:= dw_T04_EL1918.stTerminalInfo.nTerminal_State,
												sTerminalState						=> dw_T04_EL1918.stTerminalInfo.sTerminalInfo,
												bTerminalOperational				=> dw_T04_EL1918.stTerminalInfo.bTerminalOperational);
												
dw_T05_EL1918.stTerminalInfo.fbTerminalInfo(	nTerminalState						:= dw_T05_EL1918.stTerminalInfo.nTerminal_State,
												sTerminalState						=> dw_T05_EL1918.stTerminalInfo.sTerminalInfo,
												bTerminalOperational				=> dw_T05_EL1918.stTerminalInfo.bTerminalOperational);
												
dw_T06_EL2904.stTerminalInfo.fbTerminalInfo(	nTerminalState						:= dw_T06_EL2904.stTerminalInfo.nTerminal_State,
												sTerminalState						=> dw_T06_EL2904.stTerminalInfo.sTerminalInfo,
												bTerminalOperational				=> dw_T06_EL2904.stTerminalInfo.bTerminalOperational);
												
dw_T07_EL9410.stTerminalInfo.fbTerminalInfo(	nTerminalState						:= dw_T07_EL9410.stTerminalInfo.nTerminal_State,
												sTerminalState						=> dw_T07_EL9410.stTerminalInfo.sTerminalInfo,
												bTerminalOperational				=> dw_T07_EL9410.stTerminalInfo.bTerminalOperational);
											
dw_T08_EL1809.stTerminalInfo.fbTerminalInfo(	nTerminalState						:= dw_T08_EL1809.stTerminalInfo.nTerminal_State,
												sTerminalState						=> dw_T08_EL1809.stTerminalInfo.sTerminalInfo,
												bTerminalOperational				=> dw_T08_EL1809.stTerminalInfo.bTerminalOperational);
												
dw_T09_EL2809.stTerminalInfo.fbTerminalInfo(	nTerminalState						:= dw_T09_EL2809.stTerminalInfo.nTerminal_State,
												sTerminalState						=> dw_T09_EL2809.stTerminalInfo.sTerminalInfo,
												bTerminalOperational				=> dw_T09_EL2809.stTerminalInfo.bTerminalOperational);
												
												
dw_T10_EL3058.stTerminalInfo.fbTerminalInfo(	nTerminalState						:= dw_T10_EL3058.stTerminalInfo.nTerminal_State,
												sTerminalState						=> dw_T10_EL3058.stTerminalInfo.sTerminalInfo,
												bTerminalOperational				=> dw_T10_EL3058.stTerminalInfo.bTerminalOperational);
												
dw_T11_EL1918.stTerminalInfo.fbTerminalInfo(	nTerminalState						:= dw_T11_EL1918.stTerminalInfo.nTerminal_State,
												sTerminalState						=> dw_T11_EL1918.stTerminalInfo.sTerminalInfo,
												bTerminalOperational				=> dw_T11_EL1918.stTerminalInfo.bTerminalOperational);
												
dw_T12_EL6633.stTerminalInfo.fbTerminalInfo(	nTerminalState						:= dw_T12_EL6633.stTerminalInfo.nTerminal_State,
												sTerminalState						=> dw_T12_EL6633.stTerminalInfo.sTerminalInfo,
												bTerminalOperational				=> dw_T12_EL6633.stTerminalInfo.bTerminalOperational);
												
//add boxes

Probes.stTerminalInfo.fbTerminalInfo(			nTerminalState						:= Probes.stTerminalInfo.nTerminal_State,
												sTerminalState						=> Probes.stTerminalInfo.sTerminalInfo,
												bTerminalOperational				=> Probes.stTerminalInfo.bTerminalOperational);
END_ACTION

ACTION g_ACT_Manual:
tonManualMode( IN := bManualScreen, PT := T#100MS);

IF stMachineStatus.bReadyToStart THEN
	bEnableManual											:= TRUE;
ELSE bEnableManual											:= FALSE;
END_IF
	
bManualModeOffFlag										:= FALSE;



IF bManualScreen  THEN
	
	stMasterCtrl.bManualModeRequest							:= TRUE;
	
	IF (stMachineStatus.eMachineState <> E_MachineState.MANUAL_MODE) AND tonManualMode.Q THEN
				
		stMasterCtrl.bManualModeRequest							:= FALSE; 
		bManualModeOffFlag										:= TRUE;
		
	END_IF
	
ELSE 
	stMasterCtrl.bManualModeRequest							:= FALSE; 
												
END_IF
END_ACTION

ACTION h_ACT_Statistics:

stStatisticsHMI[0].sName			:= 'TEST ZONE - LH';
stStatisticsHMI[1].sName			:= 'TEST ZONE - RH';



rGoodStatistics[0]( CLK := stCycleDataNest1.bPass);
rBadStatistics[0]( CLK := stCycleDataNest1.bFail);
rGoodStatistics[1]( CLK := stCycleDataNest2.bPass);
rBadStatistics[1]( CLK := stCycleDataNest2.bFail);

IF 	rGoodStatistics[0].Q  THEN
	
	stStatisticsHMI[0].nGood		:= stStatisticsHMI[0].nGood + 1;

ELSIF 	rBadStatistics[0].Q  THEN
	
	stStatisticsHMI[0].nBad			:= stStatisticsHMI[0].nBad + 1;
		
END_IF
								


IF stStatisticsHMI[0].bResetGood THEN
	stStatisticsHMI[0].nGood		:= 0;
END_IF

IF stStatisticsHMI[0].bResetBad THEN
	stStatisticsHMI[0].nBad			:= 0;
END_IF



IF 	rGoodStatistics[1].Q  THEN
	
	stStatisticsHMI[1].nGood		:= stStatisticsHMI[1].nGood + 1;

ELSIF 	rBadStatistics[1].Q  THEN
	
	stStatisticsHMI[1].nBad			:= stStatisticsHMI[1].nBad + 1;
		
END_IF
								


IF stStatisticsHMI[1].bResetGood THEN
	stStatisticsHMI[1].nGood		:= 0;
END_IF

IF stStatisticsHMI[1].bResetBad THEN
	stStatisticsHMI[1].nBad			:= 0;
END_IF



IF (( stStatisticsHMI[0].nGood + stStatisticsHMI[0].nBad) <> 0) THEN
	
	rEfficency							:= LREAL_TO_FMTSTR(in := (DINT_TO_REAL(stStatisticsHMI[0].nGood) /( DINT_TO_REAL(stStatisticsHMI[0].nGood) + DINT_TO_REAL(stStatisticsHMI[0].nBad))) * 100.0,iPrecision := 2, bRound := TRUE);
	stStatisticsHMI[0].nEfficency		:= CONCAT(STR1 := '%', STR2 := (rEfficency));

ELSE stStatisticsHMI[0].nEfficency		:= CONCAT(STR1 := '%', STR2 := (DINT_TO_STRING(0)));
	
END_IF

IF (( stStatisticsHMI[1].nGood + stStatisticsHMI[1].nBad) <> 0) THEN
	
	rEfficency							:= LREAL_TO_FMTSTR(in := (DINT_TO_REAL(stStatisticsHMI[1].nGood) /( DINT_TO_REAL(stStatisticsHMI[1].nGood) + DINT_TO_REAL(stStatisticsHMI[1].nBad))) * 100.0,iPrecision := 2, bRound := TRUE);
	stStatisticsHMI[1].nEfficency		:= CONCAT(STR1 := '%', STR2 := (rEfficency));

ELSE stStatisticsHMI[1].nEfficency		:= CONCAT(STR1 := '%', STR2 := (DINT_TO_STRING(0)));
	
END_IF
END_ACTION

ACTION i_ACT_TwinSAFE:
	
stTwinSAFE.iSafetyErrorAcknowledge		:= dw_T04_EL1918.iResetButton;

fbScaleAirSupply( 			nRawValue						:= UINT_TO_REAL(GVL_IO.dw_T10_EL3058.iMainPressure),
							X1								:= 0,
							X2								:= 32768,
							Y1								:= 0,
							Y2								:= 10,
							
							nOutPut							=> stTwinSAFE.iAirSupplyMeasurement);

stTwinSAFE.iAirPressureMaxValue			:= nAirPressureMaxValue;
stTwinSAFE.iAirPressureMinValue			:= nAirPressureMinValue;
stTwinSAFE.iProcessDoorClosing			:= bDoorClosingFlag;
					

////////////////////////////////////////////////////////////TwinSAFE Outputs reading//////////////////////////////////////////////////////////

dw_T06_EL2904.qEnableAirSupply_PSR1								:= SEL((dw_T06_EL2904_Reading.bResult[1]=1),FALSE,TRUE);
dw_T06_EL2904.qResetAirSupply_PSR2								:= SEL((dw_T06_EL2904_Reading.bResult[2]=1),FALSE,TRUE);
dw_T06_EL2904.qLockMainDoor										:= SEL((dw_T06_EL2904_Reading.bResult[3]=1),FALSE,TRUE);
dw_T06_EL2904.qLockProcessCylinder								:= SEL((dw_T06_EL2904_Reading.bResult[4]=1),FALSE,TRUE);

dw_T06_EL2904_Reading.fbReadOutSafety06[1]( 	sNetId 			:=NetAmsIdDevice,
	                					 		nSlaveAddr 		:=1006,
					 							nSubIndex 		:=0001,
					 							nIndex 			:=16#7001 ,
					 							pDstBuf 		:=ADR(dw_T06_EL2904_Reading.bResult[1]),
					 							cbBufLen 		:=SIZEOF(dw_T06_EL2904_Reading.bResult[1]),
					 							bExecute 		:= stPuls.bFlash4Hz,
					 							tTimeout 		:= T#500MS,
					 							bBusy 			=> dw_T06_EL2904_Reading.bBusy[1],
					 							bError 			=> dw_T06_EL2904_Reading.berror[1]);
												
dw_T06_EL2904_Reading.fbReadOutSafety06[2]( 	sNetId 			:= NetAmsIdDevice,
	                					 		nSlaveAddr 		:=1006,
					 							nSubIndex 		:=0002,
					 							nIndex 			:=16#7001 ,
					 							pDstBuf 		:=ADR(dw_T06_EL2904_Reading.bResult[2]),
					 							cbBufLen 		:=SIZEOF(dw_T06_EL2904_Reading.bResult[2]),
					 							bExecute 		:= stPuls.bFlash4Hz,
					 							tTimeout 		:= T#500MS,
					 							bBusy 			=> dw_T06_EL2904_Reading.bBusy[2],
					 							bError 			=> dw_T06_EL2904_Reading.berror[2]);
												
dw_T06_EL2904_Reading.fbReadOutSafety06[3]( 	sNetId 			:=NetAmsIdDevice,
	                					 		nSlaveAddr 		:=1006,
					 							nSubIndex 		:=0003,
					 							nIndex 			:=16#7001 ,
					 							pDstBuf 		:=ADR(dw_T06_EL2904_Reading.bResult[3]),
					 							cbBufLen 		:=SIZEOF(dw_T06_EL2904_Reading.bResult[3]),
					 							bExecute 		:= stPuls.bFlash4Hz,
					 							tTimeout 		:= T#500MS,
					 							bBusy 			=> dw_T06_EL2904_Reading.bBusy[3],
					 							bError 			=> dw_T06_EL2904_Reading.berror[3]);
											
dw_T06_EL2904_Reading.fbReadOutSafety06[4]( 	sNetId 			:= NetAmsIdDevice,
	                					 		nSlaveAddr 		:=1006,
					 							nSubIndex 		:=0004,
					 							nIndex 			:=16#7001 ,
					 							pDstBuf 		:=ADR(dw_T06_EL2904_Reading.bResult[4]),
					 							cbBufLen 		:=SIZEOF(dw_T06_EL2904_Reading.bResult[4]),
					 							bExecute 		:= stPuls.bFlash4Hz,
					 							tTimeout 		:= T#500MS,
					 							bBusy 			=> dw_T06_EL2904_Reading.bBusy[4],
					 							bError 			=> dw_T06_EL2904_Reading.berror[4]);
END_ACTION

ACTION j_ACT_MachineDefinition:
rMachineDefinitionSet2(CLK := bMachineDefinitionSet1);
fMachineDefinitionSet2(CLK := bMachineDefinitionSet1);

IF rMachineDefinitionSet2.Q THEN
	
	abMachineDefinition[1]								:= FALSE;
	abMachineDefinition[2]								:= FALSE;
	abMachineDefinition[3]								:= FALSE;
	
	stMACHINE.bHeightTest								:= FALSE;
	stMACHINE.bLeakTest									:= FALSE;
	stMACHINE.bVisionTest								:= FALSE;
	stMACHINE.bPuckLocker								:= FALSE; //Renan Added 10Jul26 - Puck Locker
	stMACHINE.sName										:= '';
	stMACHINE.bMachine[1]								:= FALSE;
	stMACHINE.bMachine[2]								:= FALSE;
	stMACHINE.bMachine[3]								:= FALSE;

END_IF

IF fMachineDefinitionSet2.Q THEN

	FOR i := 1 TO 3 DO
	
		IF 	nMachineDefinitionIndex2 = i THEN
			
			abMachineDefinition[i] 						:= TRUE;
		
		END_IF
	
	END_FOR
ELSE i													:= 0;
	
END_IF


IF abMachineDefinition[1] THEN
	
	stMACHINE.bHeightTest								:= TRUE;
	stMACHINE.bLeakTest									:= NOT bOnlyHeightTestBypass;
	stMACHINE.bVisionTest								:= NOT bOnlyHeightTestBypass;
	stMACHINE.bPuckLocker								:= FALSE; //Renan Added 10Jul26 - Puck Locker
	stMACHINE.sName										:= 'LT-WH-VI LEAK TEST: FLUID PATH , HEIGHT TEST: FPB WELDING, VISION INSPECTION: EWIS FOAM';
	stMACHINE.bMachine[1]								:= TRUE;
	stMACHINE.bMachine[2]								:= FALSE;
	stMACHINE.bMachine[3]								:= FALSE;
	
	sAplication                     					:= ' Leak Test - Weld Height - Vision Inspection ';
	sSystemName											:= ' LT-WH-VI - FLUID PATH CAP ' ;

END_IF

IF abMachineDefinition[2] THEN
	
	stMACHINE.bHeightTest								:= TRUE;
	stMACHINE.bLeakTest									:= FALSE;
	stMACHINE.bVisionTest								:= NOT bOnlyHeightTestBypass;
	stMACHINE.bPuckLocker								:= TRUE; //Renan Added 10Jul26 - Puck Locker
	stMACHINE.sName										:= 'WH: HEIGHT TEST: FPB WELDING ';
	stMACHINE.bMachine[1]								:= FALSE;
	stMACHINE.bMachine[2]								:= TRUE;
	stMACHINE.bMachine[3]								:= FALSE;
	
	sAplication                     					:= ' Weld Height';
	sSystemName											:= ' WH - FLUID PATH BODY ' ;
	
END_IF

IF abMachineDefinition[3] THEN
	
	stMACHINE.bHeightTest								:= FALSE;
	stMACHINE.bLeakTest									:= TRUE;
	stMACHINE.bVisionTest								:= FALSE;
	stMACHINE.bPuckLocker								:= FALSE; //Renan Added 10Jul26 - Puck Locker
	stMACHINE.sName										:= 'LT LEAK TEST: RESERVOIR ';
	stMACHINE.bMachine[1]								:= FALSE;
	stMACHINE.bMachine[2]								:= FALSE;
	stMACHINE.bMachine[3]								:= TRUE;
	
	sAplication                     					:= ' Leak Test';
	sSystemName											:= ' LT - RESERVOIR ' ;
	
END_IF
END_ACTION

END_PROGRAM

// ---- POUs/Utilities/FB_Scale.TcPOU
FUNCTION_BLOCK FB_Scale
VAR_INPUT
	
	nRawValue									: REAL;	//Input value to scale
	X1											: REAL; // x => first point
	X2											: REAL; // x => second point
	Y1											: REAL; // y => first point
	Y2											: REAL; // y => second point
	n											: REAL; // intersection point. if there no point it will be 0


END_VAR
VAR_OUTPUT
	
	m											: REAL; // slope
	nOutPut										: UINT; // output

END_VAR
VAR
END_VAR

// Y points are from the signal that i'm scaling
	
m						:= (Y2-Y1)/(X2-X1);

nOutPut						:= REAL_TO_UINT((m*nRawValue) +n);

END_FUNCTION_BLOCK

// ---- POUs/A_MASTER/A_3_PRG_FaultHandling.TcPOU
PROGRAM A_3_PRG_FaultHandling
VAR
	

	bEventsFlag					: ARRAY [0..100] OF BOOL;
	i							: DINT;
	Counter						: CTU;			



END_VAR

a_ACT_Set_Events();
/////////////////////////////////////////////////////////////////////////////////////MASTER FAULT MONITORS////////////////////////////////////////////////////////////////////////////////////


stMasterCtrl.bNoFault 												:= 	NOT stStationEvents[0].bFault AND NOT stStationEvents[1].bFault AND
                                            							NOT stStationEvents[2].bFault AND NOT stStationEvents[3].bFault AND NOT stStationEvents[4].bFault;

stMasterCtrl.bCycleStopRequest										:= stStationEvents[0].bCycleStopRequest OR stStationEvents[1].bCycleStopRequest OR
																		stStationEvents[2].bCycleStopRequest OR stStationEvents[3].bCycleStopRequest OR stStationEvents[4].bCycleStopRequest;

ACTION a_ACT_Set_Events:
/////////////////////////////////////////////////////////////////////////////////////TwinSAFE/////////////////////////////////////////////////////////////////////////////////////

stStationEvents[0].aEvents[0].bFault						:= TRUE;
stStationEvents[0].aEvents[0].bEventFlag					:= stTwinSAFE.qAirErrorSignal;
stStationEvents[0].aEvents[0].bEventText					:= 'Pressure Error';
stStationEvents[0].aEvents[0].sSolution						:= 'Check Air Supply system';

stStationEvents[0].aEvents[1].bFault						:= TRUE;
stStationEvents[0].aEvents[1].bEventFlag					:= stTwinSAFE.qAirPressureAbove;
stStationEvents[0].aEvents[1].bEventText					:= 'System overpressurized' ;
stStationEvents[0].aEvents[1].sSolution						:= 'set the main valve to the right pressure';

stStationEvents[0].aEvents[2].bFault						:= TRUE;
stStationEvents[0].aEvents[2].bEventFlag					:= stTwinSAFE.qAirPressureBelow;
stStationEvents[0].aEvents[2].bEventText					:= 'Not enough pressure in the system' ;
stStationEvents[0].aEvents[2].sSolution						:= 'set the main valve to the right pressure and check the air supply';

stStationEvents[0].aEvents[3].bFault						:= TRUE;
stStationEvents[0].aEvents[3].bEventFlag					:= NOT dw_T04_EL1918.iEStopChannel1 AND dw_T04_EL1918.iEStopChannel2;
stStationEvents[0].aEvents[3].bEventText					:= 'E-STOP CH1 malfunction' ;
stStationEvents[0].aEvents[3].sSolution						:= 'Check E-STOP CH1';

stStationEvents[0].aEvents[4].bFault						:= TRUE;
stStationEvents[0].aEvents[4].bEventFlag					:= dw_T04_EL1918.iEStopChannel1 AND NOT dw_T04_EL1918.iEStopChannel2;
stStationEvents[0].aEvents[4].bEventText					:= 'E-STOP CH2 malfunction' ;
stStationEvents[0].aEvents[4].sSolution						:= 'Check E-STOP CH2';

stStationEvents[0].aEvents[5].bFault						:= TRUE;
stStationEvents[0].aEvents[5].bEventFlag					:= stTwinSAFE.qE_StopPressed;
stStationEvents[0].aEvents[5].bEventText					:= 'E-STOP Pressed ' ;
stStationEvents[0].aEvents[5].sSolution						:= 'Release E-STOP';

stStationEvents[0].aEvents[6].bFault						:= TRUE;
stStationEvents[0].aEvents[6].bEventFlag					:= stTwinSAFE.qSafetyOk AND NOT stTwinSAFE.qSystemSafe;
stStationEvents[0].aEvents[6].bEventText					:= 'Safe system error' ;
stStationEvents[0].aEvents[6].sSolution						:= 'Check safety elements';

stStationEvents[0].aEvents[8].bFault						:= TRUE;
stStationEvents[0].aEvents[8].bEventFlag					:= stTwinSAFE.qProcessDoorUnSafe;
stStationEvents[0].aEvents[8].bEventText					:= 'Process door movement unsafe' ;
stStationEvents[0].aEvents[8].sSolution						:= 'Reset system';

stStationEvents[0].aEvents[9].bFault						:= TRUE;
stStationEvents[0].aEvents[9].bEventFlag					:= stTwinSAFE.qTwoHandsUnsafe;
stStationEvents[0].aEvents[9].bEventText					:= 'Hands in unsafe position' ;
stStationEvents[0].aEvents[9].sSolution						:= 'Reset system';

stStationEvents[0].aEvents[10].bFault						:= TRUE;
stStationEvents[0].aEvents[10].bEventFlag					:= stTwinSAFE.qProcessCylinderUnsafe AND stTwinSAFE.qSafetyOk;
stStationEvents[0].aEvents[10].bEventText					:= 'Process cylinder Unsafe' ;
stStationEvents[0].aEvents[10].sSolution					:= 'Reset system';

stStationEvents[0].aEvents[11].bFault						:= TRUE;
stStationEvents[0].aEvents[11].bEventFlag					:= stTwinSAFE.qMainDoorUnsafe AND stTwinSAFE.qSafetyOk;
stStationEvents[0].aEvents[11].bEventText					:= 'Main Door Unsafe' ;
stStationEvents[0].aEvents[11].sSolution					:= 'Reset system';

stStationEvents[0].aEvents[13].bFault						:= TRUE;
stStationEvents[0].aEvents[13].bEventFlag					:= stTwinSAFE.qMainDoorUnsafe;
stStationEvents[0].aEvents[13].bEventText					:= 'Main door Unsafe' ;
stStationEvents[0].aEvents[13].sSolution					:= 'Close door and Reset system';

stStationEvents[0].aEvents[14].bFault						:= TRUE;
stStationEvents[0].aEvents[14].bEventTimer( IN := NOT stTwinSAFE.qSafetyOk AND (stMachineStatus.eMachineState = E_MachineState.SAFETY), PT := T#20S);
stStationEvents[0].aEvents[14].bEventFlag					:= stStationEvents[0].aEvents[14].bEventTimer.Q;
stStationEvents[0].aEvents[14].bEventText					:= 'Safe system init timeout' ;
stStationEvents[0].aEvents[14].sSolution					:= 'Check safety components, reset system';

stStationEvents[0].aEvents[15].bFault						:= TRUE;
stStationEvents[0].aEvents[15].bEventTimer(IN := stTwinSAFE.qComError OR stTwinSAFE.qFBError OR stTwinSAFE.qOtherError, PT := T#1S);
stStationEvents[0].aEvents[15].bEventFlag					:= stStationEvents[0].aEvents[15].bEventTimer.Q;
stStationEvents[0].aEvents[15].bEventText					:= 'Safety System error' ;
stStationEvents[0].aEvents[15].sSolution					:= 'Close door and Reset system';

stStationEvents[0].aEvents[16].bFault						:= TRUE;
stStationEvents[0].aEvents[16].bEventFlag					:= bRejectPartFault;
stStationEvents[0].aEvents[16].bEventText					:= 'Wrong part taken andput in the reject chute' ;
stStationEvents[0].aEvents[16].sSolution					:= 'Put parts in reject shutter and restart system';


stStationEvents[0].aEvents[18].bCycleStopRequest			:= TRUE;
stStationEvents[0].aEvents[18].bEventTimer(IN := dw_T08_EL1809.iRejectSensor, PT := T#3S);
stStationEvents[0].aEvents[18].bEventFlag					:= stStationEvents[0].aEvents[18].bEventTimer.Q;
stStationEvents[0].aEvents[18].bEventText					:= 'Reject chute full ' ;
stStationEvents[0].aEvents[18].sSolution					:= 'Empty reject shutter ';

stStationEvents[0].aEvents[19].bFault						:= TRUE;
stStationEvents[0].aEvents[19].bEventTimer(IN := NOT dw_T08_EL1809.iStopButton, PT := T#3S);
stStationEvents[0].aEvents[19].bEventFlag					:= stStationEvents[0].aEvents[19].bEventTimer.Q;
stStationEvents[0].aEvents[19].bEventText					:= 'Immediate Stop requested' ;
stStationEvents[0].aEvents[19].sSolution					:= '';





/////////////////////////////////////////////////////////////////////////////////////Cards status/////////////////////////////////////////////////////////////////////////////////////

stStationEvents[0].aEvents[20].bFault						:= TRUE;
stStationEvents[0].aEvents[20].bEventFlag					:= NOT stMachineStatus.bSystemPowerUp AND dw_T01_EK1100.stTerminalInfo.nTerminal_State <> 8;
stStationEvents[0].aEvents[20].bEventText					:= 'T01_EK1100 card in fault' ;
stStationEvents[0].aEvents[20].sSolution					:= 'Reset System';

stStationEvents[0].aEvents[21].bFault						:= TRUE;
stStationEvents[0].aEvents[21].bEventFlag					:= NOT stMachineStatus.bSystemPowerUp AND dw_T02_EL6070.stTerminalInfo.nTerminal_State <> 8;
stStationEvents[0].aEvents[21].bEventText					:= 'T02_EL6070 card in fault' ;
stStationEvents[0].aEvents[21].sSolution					:= 'Reset System';

stStationEvents[0].aEvents[22].bFault						:= TRUE;
stStationEvents[0].aEvents[22].bEventFlag					:= NOT stMachineStatus.bSystemPowerUp AND dw_T03_EL6910.stTerminalInfo.nTerminal_State <> 8;
stStationEvents[0].aEvents[22].bEventText					:= 'T03_EL6910 card in fault' ;
stStationEvents[0].aEvents[22].sSolution					:= 'Reset System';

stStationEvents[0].aEvents[23].bFault						:= TRUE;
stStationEvents[0].aEvents[23].bEventFlag					:= NOT stMachineStatus.bSystemPowerUp AND dw_T04_EL1918.stTerminalInfo.nTerminal_State <> 8;
stStationEvents[0].aEvents[23].bEventText					:= 'T04_EL1918 card in fault' ;
stStationEvents[0].aEvents[23].sSolution					:= 'Reset System';

stStationEvents[0].aEvents[24].bFault						:= TRUE;
stStationEvents[0].aEvents[24].bEventFlag					:= NOT stMachineStatus.bSystemPowerUp AND dw_T05_EL1918.stTerminalInfo.nTerminal_State <> 8;
stStationEvents[0].aEvents[24].bEventText					:= 'T05_EL1918 card in fault' ;
stStationEvents[0].aEvents[24].sSolution					:= 'Reset System';

